LIN {X -0.001,Y -382.805,Z 1558.938,A 0.000,B 0.000,C 90.000,E1 24.771} C_DIS
LIN {X -0.047,Y -376.109,Z 1558.911,A 0.000,B 0.000,C 90.000,E1 20.066} C_DIS
LIN {X -0.062,Y -373.639,Z 1558.897,A 0.000,B 0.000,C 90.000,E1 17.511} C_DIS
LIN {X -0.033,Y -368.037,Z 1558.869,A 0.000,B 0.000,C 90.000,E1 12.355} C_DIS
LIN {X 0.200,Y -366.337,Z 1558.854,A 0.000,B 0.000,C 90.000,E1 9.726} C_DIS
LIN {X 0.078,Y -361.715,Z 1558.821,A 0.000,B 0.000,C 90.000,E1 3.784} C_DIS
LIN {X -0.036,Y -360.828,Z 1558.800,A 0.000,B 0.000,C 90.000,E1 0.057} C_DIS
LIN {X -0.053,Y -359.426,Z 1558.770,A 0.000,B 0.000,C 90.000,E1 354.546} C_DIS
LIN {X 0.070,Y -358.890,Z 1558.759,A 0.000,B 0.000,C 90.000,E1 352.648} C_DIS
LIN {X -0.020,Y -359.563,Z 1558.726,A 0.000,B 0.000,C 90.000,E1 346.645} C_DIS
LIN {X 0.001,Y -361.801,Z 1558.684,A 0.000,B 0.000,C 90.000,E1 339.135} C_DIS
LIN {X -0.154,Y -362.053,Z 1558.680,A 0.000,B 0.000,C 90.000,E1 338.411} C_DIS
LIN {X 0.189,Y -365.980,Z 1558.643,A 0.000,B 0.000,C 90.000,E1 331.641} C_DIS
LIN {X 0.029,Y -366.387,Z 1558.639,A 0.000,B 0.000,C 90.000,E1 330.923} C_DIS
LIN {X -0.031,Y -371.355,Z 1558.604,A 0.000,B 0.000,C 90.000,E1 324.642} C_DIS
LIN {X -0.043,Y -371.766,Z 1558.602,A 0.000,B 0.000,C 90.000,E1 324.276} C_DIS
LIN {X 0.013,Y -377.358,Z 1558.567,A 0.000,B 0.000,C 90.000,E1 318.038} C_DIS
LIN {X 0.012,Y -378.235,Z 1558.563,A 0.000,B 0.000,C 90.000,E1 317.310} C_DIS
LIN {X 0.002,Y -383.940,Z 1558.531,A 0.000,B 0.000,C 90.000,E1 311.515} C_DIS
LIN {X 0.088,Y -384.893,Z 1558.527,A 0.000,B 0.000,C 90.000,E1 310.782} C_DIS
LIN {X 0.262,Y -390.610,Z 1558.495,A 0.000,B 0.000,C 90.000,E1 305.025} C_DIS
LIN {X 0.106,Y -391.104,Z 1558.493,A 0.000,B 0.000,C 90.000,E1 304.692} C_DIS
LIN {X 0.022,Y -391.648,Z 1558.489,A 0.000,B 0.000,C 90.000,E1 303.992} C_DIS
LIN {X -0.080,Y -396.825,Z 1558.459,A 0.000,B 0.000,C 90.000,E1 298.693} C_DIS
LIN {X -0.210,Y -397.120,Z 1558.457,A 0.000,B 0.000,C 90.000,E1 298.359} C_DIS
LIN {X -0.055,Y -401.597,Z 1558.426,A 0.000,B 0.000,C 90.000,E1 292.717} C_DIS
LIN {X 0.222,Y -404.659,Z 1558.395,A 0.000,B 0.000,C 90.000,E1 287.094} C_DIS
LIN {X -0.079,Y -404.735,Z 1558.391,A 0.000,B 0.000,C 90.000,E1 286.441} C_DIS
LIN {X 0.214,Y -406.099,Z 1558.364,A 0.000,B 0.000,C 90.000,E1 281.535} C_DIS
LIN {X -0.176,Y -406.094,Z 1558.362,A 0.000,B 0.000,C 90.000,E1 281.243} C_DIS
LIN {X -0.097,Y -405.680,Z 1558.333,A 0.000,B 0.000,C 90.000,E1 276.024} C_DIS
LIN {X -0.165,Y -405.058,Z 1558.328,A 0.000,B 0.000,C 90.000,E1 274.992} C_DIS
LIN {X -0.060,Y -403.497,Z 1558.304,A 0.000,B 0.000,C 90.000,E1 270.802} C_DIS
LIN {X -0.092,Y -403.288,Z 1558.302,A 0.000,B 0.000,C 90.000,E1 270.458} C_DIS
LIN {X 0.091,Y -398.931,Z 1558.271,A 0.000,B 0.000,C 90.000,E1 264.837} C_DIS
LIN {X -0.040,Y -393.108,Z 1558.242,A 0.000,B 0.000,C 90.000,E1 259.567} C_DIS
LIN {X -0.079,Y -392.835,Z 1558.240,A 0.000,B 0.000,C 90.000,E1 259.218} C_DIS
LIN {X 0.034,Y -385.993,Z 1558.212,A 0.000,B 0.000,C 90.000,E1 254.212} C_DIS
LIN {X -0.026,Y -385.267,Z 1558.208,A 0.000,B 0.000,C 90.000,E1 253.504} C_DIS
LIN {X -0.004,Y -384.768,Z 1558.206,A 0.000,B 0.000,C 90.000,E1 253.142} C_DIS
LIN {X 0.221,Y -377.973,Z 1558.182,A 0.000,B 0.000,C 90.000,E1 248.773} C_DIS
LIN {X -0.044,Y -376.233,Z 1558.174,A 0.000,B 0.000,C 90.000,E1 247.358} C_DIS
LIN {X 0.057,Y -374.944,Z 1558.170,A 0.000,B 0.000,C 90.000,E1 246.613} C_DIS
LIN {X -0.208,Y -368.417,Z 1558.148,A 0.000,B 0.000,C 90.000,E1 242.615} C_DIS
LIN {X 0.097,Y -366.047,Z 1558.137,A 0.000,B 0.000,C 90.000,E1 240.717} C_DIS
LIN {X 0.004,Y -359.196,Z 1558.115,A 0.000,B 0.000,C 90.000,E1 236.628} C_DIS
LIN {X 0.021,Y -355.842,Z 1558.100,A 0.000,B 0.000,C 90.000,E1 233.989} C_DIS
LIN {X -0.173,Y -348.793,Z 1558.075,A 0.000,B 0.000,C 90.000,E1 229.461} C_DIS
LIN {X -0.097,Y -346.185,Z 1558.062,A 0.000,B 0.000,C 90.000,E1 227.148} C_DIS
LIN {X -0.088,Y -345.065,Z 1558.058,A 0.000,B 0.000,C 90.000,E1 226.377} C_DIS
LIN {X 0.094,Y -338.586,Z 1558.030,A 0.000,B 0.000,C 90.000,E1 221.310} C_DIS
LIN {X 0.094,Y -336.840,Z 1558.019,A 0.000,B 0.000,C 90.000,E1 219.358} C_DIS
LIN {X 0.014,Y -330.861,Z 1557.988,A 0.000,B 0.000,C 90.000,E1 213.865} C_DIS
LIN {X 0.149,Y -329.296,Z 1557.975,A 0.000,B 0.000,C 90.000,E1 211.465} C_DIS
LIN {X -0.154,Y -324.669,Z 1557.942,A 0.000,B 0.000,C 90.000,E1 205.540} C_DIS
LIN {X 0.174,Y -323.837,Z 1557.928,A 0.000,B 0.000,C 90.000,E1 203.078} C_DIS
LIN {X -0.017,Y -321.124,Z 1557.881,A 0.000,B 0.000,C 90.000,E1 194.662} C_DIS
LIN {X 0.138,Y -320.932,Z 1557.877,A 0.000,B 0.000,C 90.000,E1 193.828} C_DIS
LIN {X -0.076,Y -321.562,Z 1557.832,A 0.000,B 0.000,C 90.000,E1 185.796} C_DIS
LIN {X -0.143,Y -324.415,Z 1557.790,A 0.000,B 0.000,C 90.000,E1 178.165} C_DIS
LIN {X -0.141,Y -325.376,Z 1557.783,A 0.000,B 0.000,C 90.000,E1 176.963} C_DIS
LIN {X -0.100,Y -329.112,Z 1557.750,A 0.000,B 0.000,C 90.000,E1 170.971} C_DIS
LIN {X 0.061,Y -334.260,Z 1557.726,A 0.000,B 0.000,C 90.000,E1 166.589} C_DIS
LIN {X 0.067,Y -335.488,Z 1557.719,A 0.000,B 0.000,C 90.000,E1 165.408} C_DIS
LIN {X 0.143,Y -340.932,Z 1557.695,A 0.000,B 0.000,C 90.000,E1 161.094} C_DIS
LIN {X -0.172,Y -342.138,Z 1557.691,A 0.000,B 0.000,C 90.000,E1 160.369} C_DIS
LIN {X -0.058,Y -347.939,Z 1557.667,A 0.000,B 0.000,C 90.000,E1 156.102} C_DIS
LIN {X -0.081,Y -354.259,Z 1557.648,A 0.000,B 0.000,C 90.000,E1 152.666} C_DIS
LIN {X -0.222,Y -361.406,Z 1557.625,A 0.000,B 0.000,C 90.000,E1 148.535} C_DIS
LIN {X 0.065,Y -368.758,Z 1557.606,A 0.000,B 0.000,C 90.000,E1 145.135} C_DIS
LIN {X 0.065,Y -377.029,Z 1557.584,A 0.000,B 0.000,C 90.000,E1 141.090} C_DIS
LIN {X -0.061,Y -383.435,Z 1557.570,A 0.000,B 0.000,C 90.000,E1 138.566} C_DIS
LIN {X -0.015,Y -385.037,Z 1557.566,A 0.000,B 0.000,C 90.000,E1 137.838} C_DIS
LIN {X -0.004,Y -394.325,Z 1557.544,A 0.000,B 0.000,C 90.000,E1 133.905} C_DIS
LIN {X 0.107,Y -399.276,Z 1557.534,A 0.000,B 0.000,C 90.000,E1 132.123} C_DIS
LIN {X 0.210,Y -400.192,Z 1557.532,A 0.000,B 0.000,C 90.000,E1 131.757} C_DIS
LIN {X -0.113,Y -409.687,Z 1557.511,A 0.000,B 0.000,C 90.000,E1 127.971} C_DIS
LIN {X 0.046,Y -415.746,Z 1557.499,A 0.000,B 0.000,C 90.000,E1 125.884} C_DIS
LIN {X 0.153,Y -425.188,Z 1557.479,A 0.000,B 0.000,C 90.000,E1 122.133} C_DIS
LIN {X 0.087,Y -430.186,Z 1557.469,A 0.000,B 0.000,C 90.000,E1 120.463} C_DIS
LIN {X 0.086,Y -431.107,Z 1557.468,A 0.000,B 0.000,C 90.000,E1 120.129} C_DIS
LIN {X 0.213,Y -432.689,Z 1557.464,A 0.000,B 0.000,C 90.000,E1 119.411} C_DIS
LIN {X 0.235,Y -547.529,Z 1557.464,A 0.000,B 0.000,C 90.000,E1 119.411} C_DIS
LIN {X 0.136,Y -547.944,Z 1557.464,A 0.000,B 0.000,C 90.000,E1 119.411} C_DIS
LIN {X -0.002,Y -549.482,Z 1557.463,A 0.000,B 0.000,C 90.000,E1 119.283} C_DIS
LIN {X -0.140,Y -550.297,Z 1557.462,A 0.000,B 0.000,C 90.000,E1 119.155} C_DIS
LIN {X -0.113,Y -551.406,Z 1557.460,A 0.000,B 0.000,C 90.000,E1 118.871} C_DIS
LIN {X 0.136,Y -552.267,Z 1557.459,A 0.000,B 0.000,C 90.000,E1 118.565} C_DIS
LIN {X -0.095,Y -552.986,Z 1557.457,A 0.000,B 0.000,C 90.000,E1 118.309} C_DIS
LIN {X 0.202,Y -554.083,Z 1557.454,A 0.000,B 0.000,C 90.000,E1 117.719} C_DIS
LIN {X 0.286,Y -555.333,Z 1557.449,A 0.000,B 0.000,C 90.000,E1 116.873} C_DIS
LIN {X 0.132,Y -556.264,Z 1557.445,A 0.000,B 0.000,C 90.000,E1 116.052} C_DIS
LIN {X 0.232,Y -556.929,Z 1557.440,A 0.000,B 0.000,C 90.000,E1 115.207} C_DIS
LIN {X 0.095,Y -557.406,Z 1557.436,A 0.000,B 0.000,C 90.000,E1 114.387} C_DIS
LIN {X 0.259,Y -557.817,Z 1557.429,A 0.000,B 0.000,C 90.000,E1 113.259} C_DIS
LIN {X 0.295,Y -558.115,Z 1557.420,A 0.000,B 0.000,C 90.000,E1 111.589} C_DIS
LIN {X 0.254,Y -558.382,Z 1557.414,A 0.000,B 0.000,C 90.000,E1 110.482} C_DIS
LIN {X 0.214,Y -558.672,Z 1557.403,A 0.000,B 0.000,C 90.000,E1 108.544} C_DIS
LIN {X 0.014,Y -559.067,Z 1557.392,A 0.000,B 0.000,C 90.000,E1 106.622} C_DIS
LIN {X 0.206,Y -559.382,Z 1557.382,A 0.000,B 0.000,C 90.000,E1 104.662} C_DIS
LIN {X -0.130,Y -559.748,Z 1557.369,A 0.000,B 0.000,C 90.000,E1 102.479} C_DIS
LIN {X -0.186,Y -560.141,Z 1557.359,A 0.000,B 0.000,C 90.000,E1 100.546} C_DIS
LIN {X 0.060,Y -560.700,Z 1557.349,A 0.000,B 0.000,C 90.000,E1 98.859} C_DIS
LIN {X 0.085,Y -561.063,Z 1557.342,A 0.000,B 0.000,C 90.000,E1 97.473} C_DIS
LIN {X -0.212,Y -561.574,Z 1557.331,A 0.000,B 0.000,C 90.000,E1 95.568} C_DIS
LIN {X -0.094,Y -562.028,Z 1557.322,A 0.000,B 0.000,C 90.000,E1 93.898} C_DIS
LIN {X 0.057,Y -562.524,Z 1557.311,A 0.000,B 0.000,C 90.000,E1 91.949} C_DIS
LIN {X 0.124,Y -562.968,Z 1557.302,A 0.000,B 0.000,C 90.000,E1 90.286} C_DIS
LIN {X -0.274,Y -563.518,Z 1557.291,A 0.000,B 0.000,C 90.000,E1 88.396} C_DIS
LIN {X 0.265,Y -563.992,Z 1557.283,A 0.000,B 0.000,C 90.000,E1 86.963} C_DIS
LIN {X -0.030,Y -564.769,Z 1557.273,A 0.000,B 0.000,C 90.000,E1 85.065} C_DIS
LIN {X 0.262,Y -565.685,Z 1557.262,A 0.000,B 0.000,C 90.000,E1 83.109} C_DIS
LIN {X -0.021,Y -566.590,Z 1557.253,A 0.000,B 0.000,C 90.000,E1 81.489} C_DIS
LIN {X 0.193,Y -567.568,Z 1557.245,A 0.000,B 0.000,C 90.000,E1 80.095} C_DIS
LIN {X -0.152,Y -569.200,Z 1557.233,A 0.000,B 0.000,C 90.000,E1 77.937} C_DIS
LIN {X 0.207,Y -570.273,Z 1557.225,A 0.000,B 0.000,C 90.000,E1 76.533} C_DIS
LIN {X 0.160,Y -571.223,Z 1557.218,A 0.000,B 0.000,C 90.000,E1 75.172} C_DIS
LIN {X -0.098,Y -572.486,Z 1557.206,A 0.000,B 0.000,C 90.000,E1 73.015} C_DIS
LIN {X -0.311,Y -573.388,Z 1557.197,A 0.000,B 0.000,C 90.000,E1 71.402} C_DIS
LIN {X 0.032,Y -574.192,Z 1557.189,A 0.000,B 0.000,C 90.000,E1 70.007} C_DIS
LIN {X -0.321,Y -575.150,Z 1557.180,A 0.000,B 0.000,C 90.000,E1 68.411} C_DIS
LIN {X -0.062,Y -576.417,Z 1557.169,A 0.000,B 0.000,C 90.000,E1 66.485} C_DIS
LIN {X 0.085,Y -577.433,Z 1557.160,A 0.000,B 0.000,C 90.000,E1 64.845} C_DIS
LIN {X 0.102,Y -578.606,Z 1557.150,A 0.000,B 0.000,C 90.000,E1 62.948} C_DIS
LIN {X 0.299,Y -579.699,Z 1557.141,A 0.000,B 0.000,C 90.000,E1 61.307} C_DIS
LIN {X 0.018,Y -580.309,Z 1557.135,A 0.000,B 0.000,C 90.000,E1 60.255} C_DIS
LIN {X -0.258,Y -580.520,Z 1557.129,A 0.000,B 0.000,C 90.000,E1 59.203} C_DIS
LIN {X -0.234,Y -580.505,Z 1557.123,A 0.000,B 0.000,C 90.000,E1 58.122} C_DIS
LIN {X -0.222,Y -580.344,Z 1557.120,A 0.000,B 0.000,C 90.000,E1 57.582} C_DIS
LIN {X -0.211,Y -579.942,Z 1557.117,A 0.000,B 0.000,C 90.000,E1 57.041} C_DIS
LIN {X -0.204,Y -579.166,Z 1557.114,A 0.000,B 0.000,C 90.000,E1 56.501} C_DIS
LIN {X -0.043,Y -578.534,Z 1557.112,A 0.000,B 0.000,C 90.000,E1 56.215} C_DIS
LIN {X -0.180,Y -577.252,Z 1557.111,A 0.000,B 0.000,C 90.000,E1 55.928} C_DIS
LIN {X 0.268,Y -576.550,Z 1557.110,A 0.000,B 0.000,C 90.000,E1 55.801} C_DIS
LIN {X -0.134,Y -575.785,Z 1557.110,A 0.000,B 0.000,C 90.000,E1 55.801} C_DIS
LIN {X -0.134,Y -442.133,Z 1557.110,A 0.000,B 0.000,C 90.000,E1 55.801} C_DIS
LIN {X 0.137,Y -433.157,Z 1557.087,A 0.000,B 0.000,C 90.000,E1 51.698} C_DIS
LIN {X -0.023,Y -431.283,Z 1557.082,A 0.000,B 0.000,C 90.000,E1 50.723} C_DIS
LIN {X -0.019,Y -422.094,Z 1557.059,A 0.000,B 0.000,C 90.000,E1 46.701} C_DIS
LIN {X 0.050,Y -418.963,Z 1557.050,A 0.000,B 0.000,C 90.000,E1 45.000} C_DIS
LIN {X -0.062,Y -418.275,Z 1557.048,A 0.000,B 0.000,C 90.000,E1 44.676} C_DIS
LIN {X 0.014,Y -408.785,Z 1557.023,A 0.000,B 0.000,C 90.000,E1 40.216} C_DIS
LIN {X 0.188,Y -405.869,Z 1557.014,A 0.000,B 0.000,C 90.000,E1 38.463} C_DIS
LIN {X -0.163,Y -397.556,Z 1556.991,A 0.000,B 0.000,C 90.000,E1 34.326} C_DIS
LIN {X 0.245,Y -393.794,Z 1556.977,A 0.000,B 0.000,C 90.000,E1 31.799} C_DIS
LIN {X -0.174,Y -386.377,Z 1556.953,A 0.000,B 0.000,C 90.000,E1 27.590} C_DIS
LIN {X -0.032,Y -382.670,Z 1556.937,A 0.000,B 0.000,C 90.000,E1 24.695} C_DIS
LIN {X -0.099,Y -376.018,Z 1556.911,A 0.000,B 0.000,C 90.000,E1 19.993} C_DIS
LIN {X 0.118,Y -373.550,Z 1556.897,A 0.000,B 0.000,C 90.000,E1 17.402} C_DIS
LIN {X 0.156,Y -367.973,Z 1556.868,A 0.000,B 0.000,C 90.000,E1 12.243} C_DIS
LIN {X 0.175,Y -366.548,Z 1556.856,A 0.000,B 0.000,C 90.000,E1 10.018} C_DIS
LIN {X -0.113,Y -365.837,Z 1556.852,A 0.000,B 0.000,C 90.000,E1 9.321} C_DIS
LIN {X -0.098,Y -361.396,Z 1556.817,A 0.000,B 0.000,C 90.000,E1 2.980} C_DIS
LIN {X -0.007,Y -360.906,Z 1556.802,A 0.000,B 0.000,C 90.000,E1 0.344} C_DIS
LIN {X 0.105,Y -360.314,Z 1556.795,A 0.000,B 0.000,C 90.000,E1 359.026} C_DIS
LIN {X -0.053,Y -359.426,Z 1556.770,A 0.000,B 0.000,C 90.000,E1 354.546} C_DIS
LIN {X 0.070,Y -358.890,Z 1556.759,A 0.000,B 0.000,C 90.000,E1 352.648} C_DIS
LIN {X -0.020,Y -359.563,Z 1556.726,A 0.000,B 0.000,C 90.000,E1 346.645} C_DIS
LIN {X 0.001,Y -361.801,Z 1556.684,A 0.000,B 0.000,C 90.000,E1 339.135} C_DIS
LIN {X -0.154,Y -362.053,Z 1556.680,A 0.000,B 0.000,C 90.000,E1 338.411} C_DIS
LIN {X 0.189,Y -365.980,Z 1556.643,A 0.000,B 0.000,C 90.000,E1 331.641} C_DIS
LIN {X 0.029,Y -366.387,Z 1556.639,A 0.000,B 0.000,C 90.000,E1 330.923} C_DIS
LIN {X -0.031,Y -371.355,Z 1556.604,A 0.000,B 0.000,C 90.000,E1 324.642} C_DIS
LIN {X -0.043,Y -371.766,Z 1556.602,A 0.000,B 0.000,C 90.000,E1 324.276} C_DIS
LIN {X 0.013,Y -377.358,Z 1556.567,A 0.000,B 0.000,C 90.000,E1 318.038} C_DIS
LIN {X 0.012,Y -378.235,Z 1556.563,A 0.000,B 0.000,C 90.000,E1 317.310} C_DIS
LIN {X 0.002,Y -383.940,Z 1556.531,A 0.000,B 0.000,C 90.000,E1 311.515} C_DIS
LIN {X 0.088,Y -384.893,Z 1556.527,A 0.000,B 0.000,C 90.000,E1 310.782} C_DIS
LIN {X 0.262,Y -390.610,Z 1556.495,A 0.000,B 0.000,C 90.000,E1 305.025} C_DIS
LIN {X 0.106,Y -391.104,Z 1556.493,A 0.000,B 0.000,C 90.000,E1 304.692} C_DIS
LIN {X 0.022,Y -391.648,Z 1556.489,A 0.000,B 0.000,C 90.000,E1 303.992} C_DIS
LIN {X -0.080,Y -396.825,Z 1556.459,A 0.000,B 0.000,C 90.000,E1 298.693} C_DIS
LIN {X -0.210,Y -397.120,Z 1556.457,A 0.000,B 0.000,C 90.000,E1 298.359} C_DIS
LIN {X -0.055,Y -401.597,Z 1556.426,A 0.000,B 0.000,C 90.000,E1 292.717} C_DIS
LIN {X 0.222,Y -404.659,Z 1556.395,A 0.000,B 0.000,C 90.000,E1 287.094} C_DIS
LIN {X -0.079,Y -404.735,Z 1556.391,A 0.000,B 0.000,C 90.000,E1 286.441} C_DIS
LIN {X 0.214,Y -406.099,Z 1556.364,A 0.000,B 0.000,C 90.000,E1 281.535} C_DIS
LIN {X -0.176,Y -406.094,Z 1556.362,A 0.000,B 0.000,C 90.000,E1 281.243} C_DIS
LIN {X -0.097,Y -405.680,Z 1556.333,A 0.000,B 0.000,C 90.000,E1 276.024} C_DIS
LIN {X -0.165,Y -405.058,Z 1556.328,A 0.000,B 0.000,C 90.000,E1 274.992} C_DIS
LIN {X -0.060,Y -403.497,Z 1556.304,A 0.000,B 0.000,C 90.000,E1 270.802} C_DIS
LIN {X -0.092,Y -403.288,Z 1556.302,A 0.000,B 0.000,C 90.000,E1 270.458} C_DIS
LIN {X 0.091,Y -398.931,Z 1556.271,A 0.000,B 0.000,C 90.000,E1 264.837} C_DIS
LIN {X -0.040,Y -393.108,Z 1556.242,A 0.000,B 0.000,C 90.000,E1 259.567} C_DIS
LIN {X -0.079,Y -392.835,Z 1556.240,A 0.000,B 0.000,C 90.000,E1 259.218} C_DIS
LIN {X 0.034,Y -385.993,Z 1556.212,A 0.000,B 0.000,C 90.000,E1 254.212} C_DIS
LIN {X -0.026,Y -385.267,Z 1556.208,A 0.000,B 0.000,C 90.000,E1 253.504} C_DIS
LIN {X -0.004,Y -384.768,Z 1556.206,A 0.000,B 0.000,C 90.000,E1 253.142} C_DIS
LIN {X 0.221,Y -377.973,Z 1556.182,A 0.000,B 0.000,C 90.000,E1 248.773} C_DIS
LIN {X -0.044,Y -376.233,Z 1556.174,A 0.000,B 0.000,C 90.000,E1 247.358} C_DIS
LIN {X 0.057,Y -374.944,Z 1556.170,A 0.000,B 0.000,C 90.000,E1 246.613} C_DIS
LIN {X -0.208,Y -368.417,Z 1556.148,A 0.000,B 0.000,C 90.000,E1 242.615} C_DIS
LIN {X 0.097,Y -366.047,Z 1556.137,A 0.000,B 0.000,C 90.000,E1 240.717} C_DIS
LIN {X 0.004,Y -359.196,Z 1556.115,A 0.000,B 0.000,C 90.000,E1 236.628} C_DIS
LIN {X 0.021,Y -355.842,Z 1556.100,A 0.000,B 0.000,C 90.000,E1 233.989} C_DIS
LIN {X -0.173,Y -348.793,Z 1556.075,A 0.000,B 0.000,C 90.000,E1 229.461} C_DIS
LIN {X -0.097,Y -346.185,Z 1556.062,A 0.000,B 0.000,C 90.000,E1 227.148} C_DIS
LIN {X -0.088,Y -345.065,Z 1556.058,A 0.000,B 0.000,C 90.000,E1 226.377} C_DIS
LIN {X 0.094,Y -338.586,Z 1556.030,A 0.000,B 0.000,C 90.000,E1 221.310} C_DIS
LIN {X 0.094,Y -336.840,Z 1556.019,A 0.000,B 0.000,C 90.000,E1 219.358} C_DIS
LIN {X 0.014,Y -330.861,Z 1555.988,A 0.000,B 0.000,C 90.000,E1 213.865} C_DIS
LIN {X 0.149,Y -329.296,Z 1555.975,A 0.000,B 0.000,C 90.000,E1 211.465} C_DIS
LIN {X -0.154,Y -324.669,Z 1555.942,A 0.000,B 0.000,C 90.000,E1 205.540} C_DIS
LIN {X 0.174,Y -323.837,Z 1555.928,A 0.000,B 0.000,C 90.000,E1 203.078} C_DIS
LIN {X -0.017,Y -321.124,Z 1555.881,A 0.000,B 0.000,C 90.000,E1 194.662} C_DIS
LIN {X 0.138,Y -320.932,Z 1555.877,A 0.000,B 0.000,C 90.000,E1 193.828} C_DIS
LIN {X -0.076,Y -321.562,Z 1555.832,A 0.000,B 0.000,C 90.000,E1 185.796} C_DIS
LIN {X -0.143,Y -324.415,Z 1555.790,A 0.000,B 0.000,C 90.000,E1 178.165} C_DIS
LIN {X -0.141,Y -325.376,Z 1555.783,A 0.000,B 0.000,C 90.000,E1 176.963} C_DIS
LIN {X -0.100,Y -329.112,Z 1555.750,A 0.000,B 0.000,C 90.000,E1 170.971} C_DIS
LIN {X 0.061,Y -334.260,Z 1555.726,A 0.000,B 0.000,C 90.000,E1 166.589} C_DIS
LIN {X 0.067,Y -335.488,Z 1555.719,A 0.000,B 0.000,C 90.000,E1 165.408} C_DIS
LIN {X 0.143,Y -340.932,Z 1555.695,A 0.000,B 0.000,C 90.000,E1 161.094} C_DIS
LIN {X -0.172,Y -342.138,Z 1555.691,A 0.000,B 0.000,C 90.000,E1 160.369} C_DIS
LIN {X -0.058,Y -347.939,Z 1555.667,A 0.000,B 0.000,C 90.000,E1 156.102} C_DIS
LIN {X -0.081,Y -354.259,Z 1555.648,A 0.000,B 0.000,C 90.000,E1 152.666} C_DIS
LIN {X -0.222,Y -361.406,Z 1555.625,A 0.000,B 0.000,C 90.000,E1 148.535} C_DIS
LIN {X 0.065,Y -368.758,Z 1555.606,A 0.000,B 0.000,C 90.000,E1 145.135} C_DIS
LIN {X 0.065,Y -377.029,Z 1555.584,A 0.000,B 0.000,C 90.000,E1 141.090} C_DIS
LIN {X -0.061,Y -383.435,Z 1555.570,A 0.000,B 0.000,C 90.000,E1 138.566} C_DIS
LIN {X -0.015,Y -385.037,Z 1555.566,A 0.000,B 0.000,C 90.000,E1 137.838} C_DIS
LIN {X -0.004,Y -394.325,Z 1555.544,A 0.000,B 0.000,C 90.000,E1 133.905} C_DIS
LIN {X 0.107,Y -399.276,Z 1555.534,A 0.000,B 0.000,C 90.000,E1 132.123} C_DIS
LIN {X 0.210,Y -400.192,Z 1555.532,A 0.000,B 0.000,C 90.000,E1 131.757} C_DIS
LIN {X -0.113,Y -409.687,Z 1555.511,A 0.000,B 0.000,C 90.000,E1 127.971} C_DIS
LIN {X 0.046,Y -415.746,Z 1555.499,A 0.000,B 0.000,C 90.000,E1 125.884} C_DIS
LIN {X 0.153,Y -425.188,Z 1555.479,A 0.000,B 0.000,C 90.000,E1 122.133} C_DIS
LIN {X -0.021,Y -429.348,Z 1555.471,A 0.000,B 0.000,C 90.000,E1 120.747} C_DIS
LIN {X -0.059,Y -547.338,Z 1555.471,A 0.000,B 0.000,C 90.000,E1 120.747} C_DIS
LIN {X 0.189,Y -547.525,Z 1555.471,A 0.000,B 0.000,C 90.000,E1 120.718} C_DIS
LIN {X 0.151,Y -549.162,Z 1555.470,A 0.000,B 0.000,C 90.000,E1 120.590} C_DIS
LIN {X 0.111,Y -549.962,Z 1555.469,A 0.000,B 0.000,C 90.000,E1 120.463} C_DIS
LIN {X -0.132,Y -551.149,Z 1555.468,A 0.000,B 0.000,C 90.000,E1 120.207} C_DIS
LIN {X -0.095,Y -552.015,Z 1555.466,A 0.000,B 0.000,C 90.000,E1 119.922} C_DIS
LIN {X 0.191,Y -553.358,Z 1555.463,A 0.000,B 0.000,C 90.000,E1 119.333} C_DIS
LIN {X 0.265,Y -554.779,Z 1555.458,A 0.000,B 0.000,C 90.000,E1 118.487} C_DIS
LIN {X 0.355,Y -555.806,Z 1555.454,A 0.000,B 0.000,C 90.000,E1 117.641} C_DIS
LIN {X -0.011,Y -556.785,Z 1555.448,A 0.000,B 0.000,C 90.000,E1 116.565} C_DIS
LIN {X -0.114,Y -557.426,Z 1555.441,A 0.000,B 0.000,C 90.000,E1 115.463} C_DIS
LIN {X 0.051,Y -557.781,Z 1555.435,A 0.000,B 0.000,C 90.000,E1 114.335} C_DIS
LIN {X 0.224,Y -558.098,Z 1555.429,A 0.000,B 0.000,C 90.000,E1 113.206} C_DIS
LIN {X -0.247,Y -558.383,Z 1555.420,A 0.000,B 0.000,C 90.000,E1 111.589} C_DIS
LIN {X 0.240,Y -558.636,Z 1555.414,A 0.000,B 0.000,C 90.000,E1 110.429} C_DIS
LIN {X 0.213,Y -558.948,Z 1555.403,A 0.000,B 0.000,C 90.000,E1 108.489} C_DIS
LIN {X 0.025,Y -559.341,Z 1555.392,A 0.000,B 0.000,C 90.000,E1 106.567} C_DIS
LIN {X -0.171,Y -559.638,Z 1555.381,A 0.000,B 0.000,C 90.000,E1 104.647} C_DIS
LIN {X 0.025,Y -560.013,Z 1555.369,A 0.000,B 0.000,C 90.000,E1 102.411} C_DIS
LIN {X 0.009,Y -560.494,Z 1555.357,A 0.000,B 0.000,C 90.000,E1 100.197} C_DIS
LIN {X 0.114,Y -560.999,Z 1555.349,A 0.000,B 0.000,C 90.000,E1 98.803} C_DIS
LIN {X 0.219,Y -561.348,Z 1555.341,A 0.000,B 0.000,C 90.000,E1 97.409} C_DIS
LIN {X -0.226,Y -561.806,Z 1555.332,A 0.000,B 0.000,C 90.000,E1 95.796} C_DIS
LIN {X -0.147,Y -562.298,Z 1555.323,A 0.000,B 0.000,C 90.000,E1 94.131} C_DIS
LIN {X -0.056,Y -562.701,Z 1555.314,A 0.000,B 0.000,C 90.000,E1 92.465} C_DIS
LIN {X 0.012,Y -563.178,Z 1555.305,A 0.000,B 0.000,C 90.000,E1 90.802} C_DIS
LIN {X 0.080,Y -563.627,Z 1555.295,A 0.000,B 0.000,C 90.000,E1 89.141} C_DIS
LIN {X 0.169,Y -564.220,Z 1555.286,A 0.000,B 0.000,C 90.000,E1 87.478} C_DIS
LIN {X -0.159,Y -564.916,Z 1555.275,A 0.000,B 0.000,C 90.000,E1 85.584} C_DIS
LIN {X 0.039,Y -565.685,Z 1555.266,A 0.000,B 0.000,C 90.000,E1 83.913} C_DIS
LIN {X -0.142,Y -566.739,Z 1555.256,A 0.000,B 0.000,C 90.000,E1 82.008} C_DIS
LIN {X -0.223,Y -568.037,Z 1555.245,A 0.000,B 0.000,C 90.000,E1 80.095} C_DIS
LIN {X 0.000,Y -569.642,Z 1555.233,A 0.000,B 0.000,C 90.000,E1 77.881} C_DIS
LIN {X 0.180,Y -570.512,Z 1555.227,A 0.000,B 0.000,C 90.000,E1 76.769} C_DIS
LIN {X -0.230,Y -571.698,Z 1555.218,A 0.000,B 0.000,C 90.000,E1 75.172} C_DIS
LIN {X 0.073,Y -572.947,Z 1555.205,A 0.000,B 0.000,C 90.000,E1 72.960} C_DIS
LIN {X 0.048,Y -573.889,Z 1555.196,A 0.000,B 0.000,C 90.000,E1 71.329} C_DIS
LIN {X -0.327,Y -574.663,Z 1555.189,A 0.000,B 0.000,C 90.000,E1 70.007} C_DIS
LIN {X 0.076,Y -575.625,Z 1555.180,A 0.000,B 0.000,C 90.000,E1 68.337} C_DIS
LIN {X 0.127,Y -576.900,Z 1555.169,A 0.000,B 0.000,C 90.000,E1 66.433} C_DIS
LIN {X -0.246,Y -577.869,Z 1555.160,A 0.000,B 0.000,C 90.000,E1 64.845} C_DIS
LIN {X 0.045,Y -579.090,Z 1555.150,A 0.000,B 0.000,C 90.000,E1 62.922} C_DIS
LIN {X -0.011,Y -580.172,Z 1555.141,A 0.000,B 0.000,C 90.000,E1 61.307} C_DIS
LIN {X 0.077,Y -581.034,Z 1555.133,A 0.000,B 0.000,C 90.000,E1 59.950} C_DIS
LIN {X -0.040,Y -581.655,Z 1555.126,A 0.000,B 0.000,C 90.000,E1 58.614} C_DIS
LIN {X -0.005,Y -582.001,Z 1555.120,A 0.000,B 0.000,C 90.000,E1 57.533} C_DIS
LIN {X 0.182,Y -581.934,Z 1555.115,A 0.000,B 0.000,C 90.000,E1 56.707} C_DIS
LIN {X -0.284,Y -581.688,Z 1555.112,A 0.000,B 0.000,C 90.000,E1 56.215} C_DIS
LIN {X -0.266,Y -581.170,Z 1555.109,A 0.000,B 0.000,C 90.000,E1 55.674} C_DIS
LIN {X -0.096,Y -580.784,Z 1555.108,A 0.000,B 0.000,C 90.000,E1 55.388} C_DIS
LIN {X 0.075,Y -580.268,Z 1555.106,A 0.000,B 0.000,C 90.000,E1 55.102} C_DIS
LIN {X -0.089,Y -579.468,Z 1555.105,A 0.000,B 0.000,C 90.000,E1 54.848} C_DIS
LIN {X 0.162,Y -578.872,Z 1555.104,A 0.000,B 0.000,C 90.000,E1 54.689} C_DIS
LIN {X 0.078,Y -577.907,Z 1555.103,A 0.000,B 0.000,C 90.000,E1 54.562} C_DIS
LIN {X 0.287,Y -576.938,Z 1555.103,A 0.000,B 0.000,C 90.000,E1 54.482} C_DIS
LIN {X 0.257,Y -576.796,Z 1555.103,A 0.000,B 0.000,C 90.000,E1 54.482} C_DIS
LIN {X 0.171,Y -439.026,Z 1555.103,A 0.000,B 0.000,C 90.000,E1 54.482} C_DIS
LIN {X -0.121,Y -431.829,Z 1555.083,A 0.000,B 0.000,C 90.000,E1 51.009} C_DIS
LIN {X 0.139,Y -431.129,Z 1555.082,A 0.000,B 0.000,C 90.000,E1 50.642} C_DIS
LIN {X 0.135,Y -421.975,Z 1555.059,A 0.000,B 0.000,C 90.000,E1 46.620} C_DIS
LIN {X 0.201,Y -418.859,Z 1555.050,A 0.000,B 0.000,C 90.000,E1 44.919} C_DIS
LIN {X -0.026,Y -417.298,Z 1555.046,A 0.000,B 0.000,C 90.000,E1 44.271} C_DIS
LIN {X 0.043,Y -408.064,Z 1555.021,A 0.000,B 0.000,C 90.000,E1 39.806} C_DIS
LIN {X -0.250,Y -405.741,Z 1555.014,A 0.000,B 0.000,C 90.000,E1 38.463} C_DIS
LIN {X -0.045,Y -397.450,Z 1554.990,A 0.000,B 0.000,C 90.000,E1 34.246} C_DIS
LIN {X -0.188,Y -393.685,Z 1554.977,A 0.000,B 0.000,C 90.000,E1 31.799} C_DIS
LIN {X -0.083,Y -386.285,Z 1554.953,A 0.000,B 0.000,C 90.000,E1 27.513} C_DIS
LIN {X 0.075,Y -383.060,Z 1554.939,A 0.000,B 0.000,C 90.000,E1 24.975} C_DIS
LIN {X 0.044,Y -381.952,Z 1554.935,A 0.000,B 0.000,C 90.000,E1 24.259} C_DIS
LIN {X -0.187,Y -375.551,Z 1554.909,A 0.000,B 0.000,C 90.000,E1 19.577} C_DIS
LIN {X 0.049,Y -373.459,Z 1554.896,A 0.000,B 0.000,C 90.000,E1 17.347} C_DIS
LIN {X 0.092,Y -367.923,Z 1554.868,A 0.000,B 0.000,C 90.000,E1 12.187} C_DIS
LIN {X 0.113,Y -366.515,Z 1554.855,A 0.000,B 0.000,C 90.000,E1 9.962} C_DIS
LIN {X 0.048,Y -361.813,Z 1554.822,A 0.000,B 0.000,C 90.000,E1 4.012} C_DIS
LIN {X -0.067,Y -360.904,Z 1554.802,A 0.000,B 0.000,C 90.000,E1 0.286} C_DIS
LIN {X -0.053,Y -359.426,Z 1554.770,A 0.000,B 0.000,C 90.000,E1 354.546} C_DIS
LIN {X 0.070,Y -358.890,Z 1554.759,A 0.000,B 0.000,C 90.000,E1 352.648} C_DIS
LIN {X -0.020,Y -359.563,Z 1554.726,A 0.000,B 0.000,C 90.000,E1 346.645} C_DIS
LIN {X 0.001,Y -361.801,Z 1554.684,A 0.000,B 0.000,C 90.000,E1 339.135} C_DIS
LIN {X -0.154,Y -362.053,Z 1554.680,A 0.000,B 0.000,C 90.000,E1 338.411} C_DIS
LIN {X 0.189,Y -365.980,Z 1554.643,A 0.000,B 0.000,C 90.000,E1 331.641} C_DIS
LIN {X 0.029,Y -366.387,Z 1554.639,A 0.000,B 0.000,C 90.000,E1 330.923} C_DIS
LIN {X -0.031,Y -371.355,Z 1554.604,A 0.000,B 0.000,C 90.000,E1 324.642} C_DIS
LIN {X -0.043,Y -371.766,Z 1554.602,A 0.000,B 0.000,C 90.000,E1 324.276} C_DIS
LIN {X 0.013,Y -377.358,Z 1554.567,A 0.000,B 0.000,C 90.000,E1 318.038} C_DIS
LIN {X 0.012,Y -378.235,Z 1554.563,A 0.000,B 0.000,C 90.000,E1 317.310} C_DIS
LIN {X 0.002,Y -383.940,Z 1554.531,A 0.000,B 0.000,C 90.000,E1 311.515} C_DIS
LIN {X 0.088,Y -384.893,Z 1554.527,A 0.000,B 0.000,C 90.000,E1 310.782} C_DIS
LIN {X 0.262,Y -390.610,Z 1554.495,A 0.000,B 0.000,C 90.000,E1 305.025} C_DIS
LIN {X 0.106,Y -391.104,Z 1554.493,A 0.000,B 0.000,C 90.000,E1 304.692} C_DIS
LIN {X 0.022,Y -391.648,Z 1554.489,A 0.000,B 0.000,C 90.000,E1 303.992} C_DIS
LIN {X -0.080,Y -396.825,Z 1554.459,A 0.000,B 0.000,C 90.000,E1 298.693} C_DIS
LIN {X -0.210,Y -397.120,Z 1554.457,A 0.000,B 0.000,C 90.000,E1 298.359} C_DIS
LIN {X -0.055,Y -401.597,Z 1554.426,A 0.000,B 0.000,C 90.000,E1 292.717} C_DIS
LIN {X 0.222,Y -404.659,Z 1554.395,A 0.000,B 0.000,C 90.000,E1 287.094} C_DIS
LIN {X -0.079,Y -404.735,Z 1554.391,A 0.000,B 0.000,C 90.000,E1 286.441} C_DIS
LIN {X 0.214,Y -406.099,Z 1554.364,A 0.000,B 0.000,C 90.000,E1 281.535} C_DIS
LIN {X -0.176,Y -406.094,Z 1554.362,A 0.000,B 0.000,C 90.000,E1 281.243} C_DIS
LIN {X -0.097,Y -405.680,Z 1554.333,A 0.000,B 0.000,C 90.000,E1 276.024} C_DIS
LIN {X -0.165,Y -405.058,Z 1554.328,A 0.000,B 0.000,C 90.000,E1 274.992} C_DIS
LIN {X -0.060,Y -403.497,Z 1554.304,A 0.000,B 0.000,C 90.000,E1 270.802} C_DIS
LIN {X -0.092,Y -403.288,Z 1554.302,A 0.000,B 0.000,C 90.000,E1 270.458} C_DIS
LIN {X 0.091,Y -398.931,Z 1554.271,A 0.000,B 0.000,C 90.000,E1 264.837} C_DIS
LIN {X -0.040,Y -393.108,Z 1554.242,A 0.000,B 0.000,C 90.000,E1 259.567} C_DIS
LIN {X -0.079,Y -392.835,Z 1554.240,A 0.000,B 0.000,C 90.000,E1 259.218} C_DIS
LIN {X 0.034,Y -385.993,Z 1554.212,A 0.000,B 0.000,C 90.000,E1 254.212} C_DIS
LIN {X -0.026,Y -385.267,Z 1554.208,A 0.000,B 0.000,C 90.000,E1 253.504} C_DIS
LIN {X -0.004,Y -384.768,Z 1554.206,A 0.000,B 0.000,C 90.000,E1 253.142} C_DIS
LIN {X 0.221,Y -377.973,Z 1554.182,A 0.000,B 0.000,C 90.000,E1 248.773} C_DIS
LIN {X -0.044,Y -376.233,Z 1554.174,A 0.000,B 0.000,C 90.000,E1 247.358} C_DIS
LIN {X 0.057,Y -374.944,Z 1554.170,A 0.000,B 0.000,C 90.000,E1 246.613} C_DIS
LIN {X -0.208,Y -368.417,Z 1554.148,A 0.000,B 0.000,C 90.000,E1 242.615} C_DIS
LIN {X 0.097,Y -366.047,Z 1554.137,A 0.000,B 0.000,C 90.000,E1 240.717} C_DIS
LIN {X 0.004,Y -359.196,Z 1554.115,A 0.000,B 0.000,C 90.000,E1 236.628} C_DIS
LIN {X 0.021,Y -355.842,Z 1554.100,A 0.000,B 0.000,C 90.000,E1 233.989} C_DIS
LIN {X -0.173,Y -348.793,Z 1554.075,A 0.000,B 0.000,C 90.000,E1 229.461} C_DIS
LIN {X -0.097,Y -346.185,Z 1554.062,A 0.000,B 0.000,C 90.000,E1 227.148} C_DIS
LIN {X -0.088,Y -345.065,Z 1554.058,A 0.000,B 0.000,C 90.000,E1 226.377} C_DIS
LIN {X 0.094,Y -338.586,Z 1554.030,A 0.000,B 0.000,C 90.000,E1 221.310} C_DIS
LIN {X 0.094,Y -336.840,Z 1554.019,A 0.000,B 0.000,C 90.000,E1 219.358} C_DIS
LIN {X 0.014,Y -330.861,Z 1553.988,A 0.000,B 0.000,C 90.000,E1 213.865} C_DIS
LIN {X 0.149,Y -329.296,Z 1553.975,A 0.000,B 0.000,C 90.000,E1 211.465} C_DIS
LIN {X -0.154,Y -324.669,Z 1553.942,A 0.000,B 0.000,C 90.000,E1 205.540} C_DIS
LIN {X 0.174,Y -323.837,Z 1553.928,A 0.000,B 0.000,C 90.000,E1 203.078} C_DIS
LIN {X -0.017,Y -321.124,Z 1553.881,A 0.000,B 0.000,C 90.000,E1 194.662} C_DIS
LIN {X 0.138,Y -320.932,Z 1553.877,A 0.000,B 0.000,C 90.000,E1 193.828} C_DIS
LIN {X -0.076,Y -321.562,Z 1553.832,A 0.000,B 0.000,C 90.000,E1 185.796} C_DIS
LIN {X -0.143,Y -324.415,Z 1553.790,A 0.000,B 0.000,C 90.000,E1 178.165} C_DIS
LIN {X -0.141,Y -325.376,Z 1553.783,A 0.000,B 0.000,C 90.000,E1 176.963} C_DIS
LIN {X -0.100,Y -329.112,Z 1553.750,A 0.000,B 0.000,C 90.000,E1 170.971} C_DIS
LIN {X 0.061,Y -334.260,Z 1553.726,A 0.000,B 0.000,C 90.000,E1 166.589} C_DIS
LIN {X 0.067,Y -335.488,Z 1553.719,A 0.000,B 0.000,C 90.000,E1 165.408} C_DIS
LIN {X 0.143,Y -340.932,Z 1553.695,A 0.000,B 0.000,C 90.000,E1 161.094} C_DIS
LIN {X -0.172,Y -342.138,Z 1553.691,A 0.000,B 0.000,C 90.000,E1 160.369} C_DIS
LIN {X -0.058,Y -347.939,Z 1553.667,A 0.000,B 0.000,C 90.000,E1 156.102} C_DIS
LIN {X -0.081,Y -354.259,Z 1553.648,A 0.000,B 0.000,C 90.000,E1 152.666} C_DIS
LIN {X -0.222,Y -361.406,Z 1553.625,A 0.000,B 0.000,C 90.000,E1 148.535} C_DIS
LIN {X 0.065,Y -368.758,Z 1553.606,A 0.000,B 0.000,C 90.000,E1 145.135} C_DIS
LIN {X 0.065,Y -377.029,Z 1553.584,A 0.000,B 0.000,C 90.000,E1 141.090} C_DIS
LIN {X -0.061,Y -383.435,Z 1553.570,A 0.000,B 0.000,C 90.000,E1 138.566} C_DIS
LIN {X -0.015,Y -385.037,Z 1553.566,A 0.000,B 0.000,C 90.000,E1 137.838} C_DIS
LIN {X -0.004,Y -394.325,Z 1553.544,A 0.000,B 0.000,C 90.000,E1 133.905} C_DIS
LIN {X 0.107,Y -399.276,Z 1553.534,A 0.000,B 0.000,C 90.000,E1 132.123} C_DIS
LIN {X 0.210,Y -400.192,Z 1553.532,A 0.000,B 0.000,C 90.000,E1 131.757} C_DIS
LIN {X -0.113,Y -409.687,Z 1553.511,A 0.000,B 0.000,C 90.000,E1 127.971} C_DIS
LIN {X 0.046,Y -415.746,Z 1553.499,A 0.000,B 0.000,C 90.000,E1 125.884} C_DIS
LIN {X 0.174,Y -425.543,Z 1553.478,A 0.000,B 0.000,C 90.000,E1 122.005} C_DIS
LIN {X 0.178,Y -547.471,Z 1553.478,A 0.000,B 0.000,C 90.000,E1 122.005} C_DIS
LIN {X 0.131,Y -547.635,Z 1553.478,A 0.000,B 0.000,C 90.000,E1 122.005} C_DIS
LIN {X 0.169,Y -549.581,Z 1553.477,A 0.000,B 0.000,C 90.000,E1 121.799} C_DIS
LIN {X 0.010,Y -550.799,Z 1553.475,A 0.000,B 0.000,C 90.000,E1 121.544} C_DIS
LIN {X 0.052,Y -551.702,Z 1553.474,A 0.000,B 0.000,C 90.000,E1 121.258} C_DIS
LIN {X -0.141,Y -553.054,Z 1553.471,A 0.000,B 0.000,C 90.000,E1 120.718} C_DIS
LIN {X 0.152,Y -554.079,Z 1553.468,A 0.000,B 0.000,C 90.000,E1 120.129} C_DIS
LIN {X 0.234,Y -555.255,Z 1553.463,A 0.000,B 0.000,C 90.000,E1 119.283} C_DIS
LIN {X 0.116,Y -556.362,Z 1553.457,A 0.000,B 0.000,C 90.000,E1 118.180} C_DIS
LIN {X 0.016,Y -557.060,Z 1553.450,A 0.000,B 0.000,C 90.000,E1 117.078} C_DIS
LIN {X -0.081,Y -557.536,Z 1553.444,A 0.000,B 0.000,C 90.000,E1 115.976} C_DIS
LIN {X -0.210,Y -557.849,Z 1553.440,A 0.000,B 0.000,C 90.000,E1 115.155} C_DIS
LIN {X -0.246,Y -558.257,Z 1553.432,A 0.000,B 0.000,C 90.000,E1 113.770} C_DIS
LIN {X 0.234,Y -558.498,Z 1553.424,A 0.000,B 0.000,C 90.000,E1 112.333} C_DIS
LIN {X -0.131,Y -558.889,Z 1553.413,A 0.000,B 0.000,C 90.000,E1 110.429} C_DIS
LIN {X -0.152,Y -559.222,Z 1553.403,A 0.000,B 0.000,C 90.000,E1 108.489} C_DIS
LIN {X 0.069,Y -559.552,Z 1553.393,A 0.000,B 0.000,C 90.000,E1 106.804} C_DIS
LIN {X 0.132,Y -559.780,Z 1553.384,A 0.000,B 0.000,C 90.000,E1 105.134} C_DIS
LIN {X -0.236,Y -559.949,Z 1553.378,A 0.000,B 0.000,C 90.000,E1 104.064} C_DIS
LIN {X -0.171,Y -560.333,Z 1553.367,A 0.000,B 0.000,C 90.000,E1 102.119} C_DIS
LIN {X 0.123,Y -561.112,Z 1553.352,A 0.000,B 0.000,C 90.000,E1 99.321} C_DIS
LIN {X 0.081,Y -561.468,Z 1553.346,A 0.000,B 0.000,C 90.000,E1 98.219} C_DIS
LIN {X -0.217,Y -562.008,Z 1553.335,A 0.000,B 0.000,C 90.000,E1 96.315} C_DIS
LIN {X -0.090,Y -562.475,Z 1553.326,A 0.000,B 0.000,C 90.000,E1 94.645} C_DIS
LIN {X -0.230,Y -562.787,Z 1553.320,A 0.000,B 0.000,C 90.000,E1 93.555} C_DIS
LIN {X -0.036,Y -563.272,Z 1553.309,A 0.000,B 0.000,C 90.000,E1 91.604} C_DIS
LIN {X -0.077,Y -563.694,Z 1553.301,A 0.000,B 0.000,C 90.000,E1 90.229} C_DIS
LIN {X 0.232,Y -564.422,Z 1553.289,A 0.000,B 0.000,C 90.000,E1 87.993} C_DIS
LIN {X -0.120,Y -565.079,Z 1553.278,A 0.000,B 0.000,C 90.000,E1 86.102} C_DIS
LIN {X 0.175,Y -565.962,Z 1553.268,A 0.000,B 0.000,C 90.000,E1 84.147} C_DIS
LIN {X -0.009,Y -567.014,Z 1553.257,A 0.000,B 0.000,C 90.000,E1 82.243} C_DIS
LIN {X 0.088,Y -568.495,Z 1553.245,A 0.000,B 0.000,C 90.000,E1 80.038} C_DIS
LIN {X 0.137,Y -569.841,Z 1553.234,A 0.000,B 0.000,C 90.000,E1 78.117} C_DIS
LIN {X -0.237,Y -570.762,Z 1553.228,A 0.000,B 0.000,C 90.000,E1 77.061} C_DIS
LIN {X -0.086,Y -571.986,Z 1553.219,A 0.000,B 0.000,C 90.000,E1 75.408} C_DIS
LIN {X 0.053,Y -572.748,Z 1553.211,A 0.000,B 0.000,C 90.000,E1 74.031} C_DIS
LIN {X -0.146,Y -573.719,Z 1553.202,A 0.000,B 0.000,C 90.000,E1 72.417} C_DIS
LIN {X -0.152,Y -574.377,Z 1553.196,A 0.000,B 0.000,C 90.000,E1 71.329} C_DIS
LIN {X 0.218,Y -575.126,Z 1553.189,A 0.000,B 0.000,C 90.000,E1 69.934} C_DIS
LIN {X -0.106,Y -576.091,Z 1553.180,A 0.000,B 0.000,C 90.000,E1 68.337} C_DIS
LIN {X -0.044,Y -577.366,Z 1553.169,A 0.000,B 0.000,C 90.000,E1 66.433} C_DIS
LIN {X -0.030,Y -578.461,Z 1553.159,A 0.000,B 0.000,C 90.000,E1 64.537} C_DIS
LIN {X -0.106,Y -579.558,Z 1553.150,A 0.000,B 0.000,C 90.000,E1 62.922} C_DIS
LIN {X -0.154,Y -580.628,Z 1553.141,A 0.000,B 0.000,C 90.000,E1 61.307} C_DIS
LIN {X -0.057,Y -581.476,Z 1553.133,A 0.000,B 0.000,C 90.000,E1 59.950} C_DIS
LIN {X 0.020,Y -582.825,Z 1553.121,A 0.000,B 0.000,C 90.000,E1 57.788} C_DIS
LIN {X -0.098,Y -583.191,Z 1553.117,A 0.000,B 0.000,C 90.000,E1 56.993} C_DIS
LIN {X 0.102,Y -583.329,Z 1553.112,A 0.000,B 0.000,C 90.000,E1 56.167} C_DIS
LIN {X -0.178,Y -583.151,Z 1553.108,A 0.000,B 0.000,C 90.000,E1 55.388} C_DIS
LIN {X 0.180,Y -582.790,Z 1553.105,A 0.000,B 0.000,C 90.000,E1 54.815} C_DIS
LIN {X 0.198,Y -582.038,Z 1553.102,A 0.000,B 0.000,C 90.000,E1 54.276} C_DIS
LIN {X -0.096,Y -581.546,Z 1553.100,A 0.000,B 0.000,C 90.000,E1 54.036} C_DIS
LIN {X -0.264,Y -580.882,Z 1553.099,A 0.000,B 0.000,C 90.000,E1 53.783} C_DIS
LIN {X -0.046,Y -579.685,Z 1553.097,A 0.000,B 0.000,C 90.000,E1 53.463} C_DIS
LIN {X 0.024,Y -578.731,Z 1553.096,A 0.000,B 0.000,C 90.000,E1 53.336} C_DIS
LIN {X 0.065,Y -578.046,Z 1553.096,A 0.000,B 0.000,C 90.000,E1 53.290} C_DIS
LIN {X -0.029,Y -577.658,Z 1553.096,A 0.000,B 0.000,C 90.000,E1 53.290} C_DIS
LIN {X -0.046,Y -436.309,Z 1553.096,A 0.000,B 0.000,C 90.000,E1 53.290} C_DIS
LIN {X 0.113,Y -431.662,Z 1553.083,A 0.000,B 0.000,C 90.000,E1 50.884} C_DIS
LIN {X 0.101,Y -427.587,Z 1553.074,A 0.000,B 0.000,C 90.000,E1 49.218} C_DIS
LIN {X 0.091,Y -418.693,Z 1553.049,A 0.000,B 0.000,C 90.000,E1 44.838} C_DIS
LIN {X 0.030,Y -409.762,Z 1553.026,A 0.000,B 0.000,C 90.000,E1 40.744} C_DIS
LIN {X 0.053,Y -406.171,Z 1553.015,A 0.000,B 0.000,C 90.000,E1 38.669} C_DIS
LIN {X 0.087,Y -404.738,Z 1553.011,A 0.000,B 0.000,C 90.000,E1 37.971} C_DIS
LIN {X -0.105,Y -396.143,Z 1552.986,A 0.000,B 0.000,C 90.000,E1 33.452} C_DIS
LIN {X 0.135,Y -394.058,Z 1552.978,A 0.000,B 0.000,C 90.000,E1 32.005} C_DIS
LIN {X 0.001,Y -393.484,Z 1552.976,A 0.000,B 0.000,C 90.000,E1 31.671} C_DIS
LIN {X 0.097,Y -386.139,Z 1552.952,A 0.000,B 0.000,C 90.000,E1 27.385} C_DIS
LIN {X -0.097,Y -382.946,Z 1552.938,A 0.000,B 0.000,C 90.000,E1 24.899} C_DIS
LIN {X 0.002,Y -376.239,Z 1552.912,A 0.000,B 0.000,C 90.000,E1 20.174} C_DIS
LIN {X -0.134,Y -373.734,Z 1552.898,A 0.000,B 0.000,C 90.000,E1 17.638} C_DIS
LIN {X 0.110,Y -371.874,Z 1552.890,A 0.000,B 0.000,C 90.000,E1 16.134} C_DIS
LIN {X 0.087,Y -366.859,Z 1552.859,A 0.000,B 0.000,C 90.000,E1 10.602} C_DIS
LIN {X 0.164,Y -366.454,Z 1552.855,A 0.000,B 0.000,C 90.000,E1 9.849} C_DIS
LIN {X 0.101,Y -361.766,Z 1552.822,A 0.000,B 0.000,C 90.000,E1 3.898} C_DIS
LIN {X -0.013,Y -360.890,Z 1552.801,A 0.000,B 0.000,C 90.000,E1 0.172} C_DIS
LIN {X -0.053,Y -359.426,Z 1552.770,A 0.000,B 0.000,C 90.000,E1 354.546} C_DIS
LIN {X 0.070,Y -358.890,Z 1552.759,A 0.000,B 0.000,C 90.000,E1 352.648} C_DIS
LIN {X -0.020,Y -359.563,Z 1552.726,A 0.000,B 0.000,C 90.000,E1 346.645} C_DIS
LIN {X 0.001,Y -361.801,Z 1552.684,A 0.000,B 0.000,C 90.000,E1 339.135} C_DIS
LIN {X -0.154,Y -362.053,Z 1552.680,A 0.000,B 0.000,C 90.000,E1 338.411} C_DIS
LIN {X 0.189,Y -365.980,Z 1552.643,A 0.000,B 0.000,C 90.000,E1 331.641} C_DIS
LIN {X 0.029,Y -366.387,Z 1552.639,A 0.000,B 0.000,C 90.000,E1 330.923} C_DIS
LIN {X -0.031,Y -371.355,Z 1552.604,A 0.000,B 0.000,C 90.000,E1 324.642} C_DIS
LIN {X -0.043,Y -371.766,Z 1552.602,A 0.000,B 0.000,C 90.000,E1 324.276} C_DIS
LIN {X 0.013,Y -377.358,Z 1552.567,A 0.000,B 0.000,C 90.000,E1 318.038} C_DIS
LIN {X 0.012,Y -378.235,Z 1552.563,A 0.000,B 0.000,C 90.000,E1 317.310} C_DIS
LIN {X 0.002,Y -383.940,Z 1552.531,A 0.000,B 0.000,C 90.000,E1 311.515} C_DIS
LIN {X 0.088,Y -384.893,Z 1552.527,A 0.000,B 0.000,C 90.000,E1 310.782} C_DIS
LIN {X 0.262,Y -390.610,Z 1552.495,A 0.000,B 0.000,C 90.000,E1 305.025} C_DIS
LIN {X 0.106,Y -391.104,Z 1552.493,A 0.000,B 0.000,C 90.000,E1 304.692} C_DIS
LIN {X 0.022,Y -391.648,Z 1552.489,A 0.000,B 0.000,C 90.000,E1 303.992} C_DIS
LIN {X -0.080,Y -396.825,Z 1552.459,A 0.000,B 0.000,C 90.000,E1 298.693} C_DIS
LIN {X -0.210,Y -397.120,Z 1552.457,A 0.000,B 0.000,C 90.000,E1 298.359} C_DIS
LIN {X -0.055,Y -401.597,Z 1552.426,A 0.000,B 0.000,C 90.000,E1 292.717} C_DIS
LIN {X 0.222,Y -404.659,Z 1552.395,A 0.000,B 0.000,C 90.000,E1 287.094} C_DIS
LIN {X -0.079,Y -404.735,Z 1552.391,A 0.000,B 0.000,C 90.000,E1 286.441} C_DIS
LIN {X 0.214,Y -406.099,Z 1552.364,A 0.000,B 0.000,C 90.000,E1 281.535} C_DIS
LIN {X -0.176,Y -406.094,Z 1552.362,A 0.000,B 0.000,C 90.000,E1 281.243} C_DIS
LIN {X -0.097,Y -405.680,Z 1552.333,A 0.000,B 0.000,C 90.000,E1 276.024} C_DIS
LIN {X -0.165,Y -405.058,Z 1552.328,A 0.000,B 0.000,C 90.000,E1 274.992} C_DIS
LIN {X -0.060,Y -403.497,Z 1552.304,A 0.000,B 0.000,C 90.000,E1 270.802} C_DIS
LIN {X -0.092,Y -403.288,Z 1552.302,A 0.000,B 0.000,C 90.000,E1 270.458} C_DIS
LIN {X 0.091,Y -398.931,Z 1552.271,A 0.000,B 0.000,C 90.000,E1 264.837} C_DIS
LIN {X -0.040,Y -393.108,Z 1552.242,A 0.000,B 0.000,C 90.000,E1 259.567} C_DIS
LIN {X -0.079,Y -392.835,Z 1552.240,A 0.000,B 0.000,C 90.000,E1 259.218} C_DIS
LIN {X 0.034,Y -385.993,Z 1552.212,A 0.000,B 0.000,C 90.000,E1 254.212} C_DIS
LIN {X -0.026,Y -385.267,Z 1552.208,A 0.000,B 0.000,C 90.000,E1 253.504} C_DIS
LIN {X -0.004,Y -384.768,Z 1552.206,A 0.000,B 0.000,C 90.000,E1 253.142} C_DIS
LIN {X 0.221,Y -377.973,Z 1552.182,A 0.000,B 0.000,C 90.000,E1 248.773} C_DIS
LIN {X -0.044,Y -376.233,Z 1552.174,A 0.000,B 0.000,C 90.000,E1 247.358} C_DIS
LIN {X 0.057,Y -374.944,Z 1552.170,A 0.000,B 0.000,C 90.000,E1 246.613} C_DIS
LIN {X -0.208,Y -368.417,Z 1552.148,A 0.000,B 0.000,C 90.000,E1 242.615} C_DIS
LIN {X 0.097,Y -366.047,Z 1552.137,A 0.000,B 0.000,C 90.000,E1 240.717} C_DIS
LIN {X 0.004,Y -359.196,Z 1552.115,A 0.000,B 0.000,C 90.000,E1 236.628} C_DIS
LIN {X 0.021,Y -355.842,Z 1552.100,A 0.000,B 0.000,C 90.000,E1 233.989} C_DIS
LIN {X -0.173,Y -348.793,Z 1552.075,A 0.000,B 0.000,C 90.000,E1 229.461} C_DIS
LIN {X -0.097,Y -346.185,Z 1552.062,A 0.000,B 0.000,C 90.000,E1 227.148} C_DIS
LIN {X -0.088,Y -345.065,Z 1552.058,A 0.000,B 0.000,C 90.000,E1 226.377} C_DIS
LIN {X 0.094,Y -338.586,Z 1552.030,A 0.000,B 0.000,C 90.000,E1 221.310} C_DIS
LIN {X 0.094,Y -336.840,Z 1552.019,A 0.000,B 0.000,C 90.000,E1 219.358} C_DIS
LIN {X 0.014,Y -330.861,Z 1551.988,A 0.000,B 0.000,C 90.000,E1 213.865} C_DIS
LIN {X 0.149,Y -329.296,Z 1551.975,A 0.000,B 0.000,C 90.000,E1 211.465} C_DIS
LIN {X -0.154,Y -324.669,Z 1551.942,A 0.000,B 0.000,C 90.000,E1 205.540} C_DIS
LIN {X 0.174,Y -323.837,Z 1551.928,A 0.000,B 0.000,C 90.000,E1 203.078} C_DIS
LIN {X -0.017,Y -321.124,Z 1551.881,A 0.000,B 0.000,C 90.000,E1 194.662} C_DIS
LIN {X 0.138,Y -320.932,Z 1551.877,A 0.000,B 0.000,C 90.000,E1 193.828} C_DIS
LIN {X -0.076,Y -321.562,Z 1551.832,A 0.000,B 0.000,C 90.000,E1 185.796} C_DIS
LIN {X -0.143,Y -324.415,Z 1551.790,A 0.000,B 0.000,C 90.000,E1 178.165} C_DIS
LIN {X -0.141,Y -325.376,Z 1551.783,A 0.000,B 0.000,C 90.000,E1 176.963} C_DIS
LIN {X -0.100,Y -329.112,Z 1551.750,A 0.000,B 0.000,C 90.000,E1 170.971} C_DIS
LIN {X 0.061,Y -334.260,Z 1551.726,A 0.000,B 0.000,C 90.000,E1 166.589} C_DIS
LIN {X 0.067,Y -335.488,Z 1551.719,A 0.000,B 0.000,C 90.000,E1 165.408} C_DIS
LIN {X 0.143,Y -340.932,Z 1551.695,A 0.000,B 0.000,C 90.000,E1 161.094} C_DIS
LIN {X -0.172,Y -342.138,Z 1551.691,A 0.000,B 0.000,C 90.000,E1 160.369} C_DIS
LIN {X -0.058,Y -347.939,Z 1551.667,A 0.000,B 0.000,C 90.000,E1 156.102} C_DIS
LIN {X -0.081,Y -354.259,Z 1551.648,A 0.000,B 0.000,C 90.000,E1 152.666} C_DIS
LIN {X -0.222,Y -361.406,Z 1551.625,A 0.000,B 0.000,C 90.000,E1 148.535} C_DIS
LIN {X 0.065,Y -368.758,Z 1551.606,A 0.000,B 0.000,C 90.000,E1 145.135} C_DIS
LIN {X 0.065,Y -377.029,Z 1551.584,A 0.000,B 0.000,C 90.000,E1 141.090} C_DIS
LIN {X -0.061,Y -383.435,Z 1551.570,A 0.000,B 0.000,C 90.000,E1 138.566} C_DIS
LIN {X -0.015,Y -385.037,Z 1551.566,A 0.000,B 0.000,C 90.000,E1 137.838} C_DIS
LIN {X -0.004,Y -394.325,Z 1551.544,A 0.000,B 0.000,C 90.000,E1 133.905} C_DIS
LIN {X 0.107,Y -399.276,Z 1551.534,A 0.000,B 0.000,C 90.000,E1 132.123} C_DIS
LIN {X 0.210,Y -400.192,Z 1551.532,A 0.000,B 0.000,C 90.000,E1 131.757} C_DIS
LIN {X -0.113,Y -409.687,Z 1551.511,A 0.000,B 0.000,C 90.000,E1 127.971} C_DIS
LIN {X 0.046,Y -415.746,Z 1551.499,A 0.000,B 0.000,C 90.000,E1 125.884} C_DIS
LIN {X -0.072,Y -422.096,Z 1551.485,A 0.000,B 0.000,C 90.000,E1 123.293} C_DIS
LIN {X -0.144,Y -547.424,Z 1551.485,A 0.000,B 0.000,C 90.000,E1 123.293} C_DIS
LIN {X 0.014,Y -548.998,Z 1551.484,A 0.000,B 0.000,C 90.000,E1 123.166} C_DIS
LIN {X -0.069,Y -550.262,Z 1551.483,A 0.000,B 0.000,C 90.000,E1 122.959} C_DIS
LIN {X -0.024,Y -551.324,Z 1551.482,A 0.000,B 0.000,C 90.000,E1 122.673} C_DIS
LIN {X -0.271,Y -552.109,Z 1551.480,A 0.000,B 0.000,C 90.000,E1 122.418} C_DIS
LIN {X 0.304,Y -553.296,Z 1551.477,A 0.000,B 0.000,C 90.000,E1 121.799} C_DIS
LIN {X -0.106,Y -554.570,Z 1551.472,A 0.000,B 0.000,C 90.000,E1 121.003} C_DIS
LIN {X 0.258,Y -555.539,Z 1551.468,A 0.000,B 0.000,C 90.000,E1 120.129} C_DIS
LIN {X 0.138,Y -556.475,Z 1551.461,A 0.000,B 0.000,C 90.000,E1 119.027} C_DIS
LIN {X 0.300,Y -557.062,Z 1551.455,A 0.000,B 0.000,C 90.000,E1 117.897} C_DIS
LIN {X -0.012,Y -557.583,Z 1551.448,A 0.000,B 0.000,C 90.000,E1 116.539} C_DIS
LIN {X 0.150,Y -558.063,Z 1551.441,A 0.000,B 0.000,C 90.000,E1 115.412} C_DIS
LIN {X -0.091,Y -558.535,Z 1551.432,A 0.000,B 0.000,C 90.000,E1 113.770} C_DIS
LIN {X 0.180,Y -558.793,Z 1551.423,A 0.000,B 0.000,C 90.000,E1 112.078} C_DIS
LIN {X 0.035,Y -559.128,Z 1551.414,A 0.000,B 0.000,C 90.000,E1 110.429} C_DIS
LIN {X 0.020,Y -559.461,Z 1551.403,A 0.000,B 0.000,C 90.000,E1 108.489} C_DIS
LIN {X -0.290,Y -559.791,Z 1551.394,A 0.000,B 0.000,C 90.000,E1 106.858} C_DIS
LIN {X -0.083,Y -560.055,Z 1551.383,A 0.000,B 0.000,C 90.000,E1 104.898} C_DIS
LIN {X -0.301,Y -560.217,Z 1551.375,A 0.000,B 0.000,C 90.000,E1 103.536} C_DIS
LIN {X 0.169,Y -560.625,Z 1551.366,A 0.000,B 0.000,C 90.000,E1 101.827} C_DIS
LIN {X -0.230,Y -561.365,Z 1551.352,A 0.000,B 0.000,C 90.000,E1 99.378} C_DIS
LIN {X -0.200,Y -561.770,Z 1551.344,A 0.000,B 0.000,C 90.000,E1 97.992} C_DIS
LIN {X 0.079,Y -562.345,Z 1551.334,A 0.000,B 0.000,C 90.000,E1 96.030} C_DIS
LIN {X 0.222,Y -562.843,Z 1551.324,A 0.000,B 0.000,C 90.000,E1 94.359} C_DIS
LIN {X 0.091,Y -563.153,Z 1551.318,A 0.000,B 0.000,C 90.000,E1 93.269} C_DIS
LIN {X -0.267,Y -563.641,Z 1551.307,A 0.000,B 0.000,C 90.000,E1 91.375} C_DIS
LIN {X 0.265,Y -564.090,Z 1551.300,A 0.000,B 0.000,C 90.000,E1 89.943} C_DIS
LIN {X 0.020,Y -564.872,Z 1551.288,A 0.000,B 0.000,C 90.000,E1 87.764} C_DIS
LIN {X 0.278,Y -565.555,Z 1551.277,A 0.000,B 0.000,C 90.000,E1 85.812} C_DIS
LIN {X 0.134,Y -566.570,Z 1551.265,A 0.000,B 0.000,C 90.000,E1 83.628} C_DIS
LIN {X -0.038,Y -567.684,Z 1551.254,A 0.000,B 0.000,C 90.000,E1 81.724} C_DIS
LIN {X -0.009,Y -569.064,Z 1551.243,A 0.000,B 0.000,C 90.000,E1 79.803} C_DIS
LIN {X 0.056,Y -570.467,Z 1551.233,A 0.000,B 0.000,C 90.000,E1 77.881} C_DIS
LIN {X 0.014,Y -571.543,Z 1551.225,A 0.000,B 0.000,C 90.000,E1 76.520} C_DIS
LIN {X -0.144,Y -572.565,Z 1551.218,A 0.000,B 0.000,C 90.000,E1 75.172} C_DIS
LIN {X -0.170,Y -573.681,Z 1551.207,A 0.000,B 0.000,C 90.000,E1 73.268} C_DIS
LIN {X -0.186,Y -574.671,Z 1551.198,A 0.000,B 0.000,C 90.000,E1 71.638} C_DIS
LIN {X -0.182,Y -575.556,Z 1551.189,A 0.000,B 0.000,C 90.000,E1 70.007} C_DIS
LIN {X -0.132,Y -576.696,Z 1551.178,A 0.000,B 0.000,C 90.000,E1 68.103} C_DIS
LIN {X 0.164,Y -577.913,Z 1551.168,A 0.000,B 0.000,C 90.000,E1 66.177} C_DIS
LIN {X 0.196,Y -579.007,Z 1551.157,A 0.000,B 0.000,C 90.000,E1 64.280} C_DIS
LIN {X 0.133,Y -580.123,Z 1551.148,A 0.000,B 0.000,C 90.000,E1 62.666} C_DIS
LIN {X 0.093,Y -580.836,Z 1551.142,A 0.000,B 0.000,C 90.000,E1 61.591} C_DIS
LIN {X -0.167,Y -581.884,Z 1551.133,A 0.000,B 0.000,C 90.000,E1 59.999} C_DIS
LIN {X -0.207,Y -583.453,Z 1551.120,A 0.000,B 0.000,C 90.000,E1 57.582} C_DIS
LIN {X -0.144,Y -584.141,Z 1551.114,A 0.000,B 0.000,C 90.000,E1 56.501} C_DIS
LIN {X 0.068,Y -584.429,Z 1551.109,A 0.000,B 0.000,C 90.000,E1 55.674} C_DIS
LIN {X -0.196,Y -584.472,Z 1551.105,A 0.000,B 0.000,C 90.000,E1 54.895} C_DIS
LIN {X 0.198,Y -583.895,Z 1551.099,A 0.000,B 0.000,C 90.000,E1 53.783} C_DIS
LIN {X -0.089,Y -583.656,Z 1551.097,A 0.000,B 0.000,C 90.000,E1 53.543} C_DIS
LIN {X -0.073,Y -582.828,Z 1551.094,A 0.000,B 0.000,C 90.000,E1 53.004} C_DIS
LIN {X 0.105,Y -582.198,Z 1551.093,A 0.000,B 0.000,C 90.000,E1 52.718} C_DIS
LIN {X -0.179,Y -581.321,Z 1551.091,A 0.000,B 0.000,C 90.000,E1 52.477} C_DIS
LIN {X 0.087,Y -580.692,Z 1551.091,A 0.000,B 0.000,C 90.000,E1 52.316} C_DIS
LIN {X -0.003,Y -579.679,Z 1551.090,A 0.000,B 0.000,C 90.000,E1 52.190} C_DIS
LIN {X 0.211,Y -578.674,Z 1551.090,A 0.000,B 0.000,C 90.000,E1 52.110} C_DIS
LIN {X 0.179,Y -578.524,Z 1551.090,A 0.000,B 0.000,C 90.000,E1 52.110} C_DIS
LIN {X 0.111,Y -433.942,Z 1551.090,A 0.000,B 0.000,C 90.000,E1 52.110} C_DIS
LIN {X -0.030,Y -431.708,Z 1551.083,A 0.000,B 0.000,C 90.000,E1 50.928} C_DIS
LIN {X -0.122,Y -430.101,Z 1551.079,A 0.000,B 0.000,C 90.000,E1 50.275} C_DIS
LIN {X 0.012,Y -420.551,Z 1551.055,A 0.000,B 0.000,C 90.000,E1 45.891} C_DIS
LIN {X -0.015,Y -418.739,Z 1551.049,A 0.000,B 0.000,C 90.000,E1 44.879} C_DIS
LIN {X -0.048,Y -409.812,Z 1551.027,A 0.000,B 0.000,C 90.000,E1 40.782} C_DIS
LIN {X -0.013,Y -406.213,Z 1551.015,A 0.000,B 0.000,C 90.000,E1 38.705} C_DIS
LIN {X -0.186,Y -405.578,Z 1551.013,A 0.000,B 0.000,C 90.000,E1 38.382} C_DIS
LIN {X -0.122,Y -396.749,Z 1550.988,A 0.000,B 0.000,C 90.000,E1 33.833} C_DIS
LIN {X 0.187,Y -393.538,Z 1550.976,A 0.000,B 0.000,C 90.000,E1 31.671} C_DIS
LIN {X -0.060,Y -386.179,Z 1550.952,A 0.000,B 0.000,C 90.000,E1 27.436} C_DIS
LIN {X 0.087,Y -382.976,Z 1550.938,A 0.000,B 0.000,C 90.000,E1 24.899} C_DIS
LIN {X 0.068,Y -376.694,Z 1550.914,A 0.000,B 0.000,C 90.000,E1 20.556} C_DIS
LIN {X 0.050,Y -373.757,Z 1550.898,A 0.000,B 0.000,C 90.000,E1 17.638} C_DIS
LIN {X -0.003,Y -372.857,Z 1550.894,A 0.000,B 0.000,C 90.000,E1 16.913} C_DIS
LIN {X -0.100,Y -367.593,Z 1550.865,A 0.000,B 0.000,C 90.000,E1 11.771} C_DIS
LIN {X -0.016,Y -366.474,Z 1550.855,A 0.000,B 0.000,C 90.000,E1 9.905} C_DIS
LIN {X -0.078,Y -361.779,Z 1550.822,A 0.000,B 0.000,C 90.000,E1 3.955} C_DIS
LIN {X 0.167,Y -360.897,Z 1550.801,A 0.000,B 0.000,C 90.000,E1 0.172} C_DIS
LIN {X -0.053,Y -359.426,Z 1550.770,A 0.000,B 0.000,C 90.000,E1 354.546} C_DIS
LIN {X 0.070,Y -358.890,Z 1550.759,A 0.000,B 0.000,C 90.000,E1 352.648} C_DIS
LIN {X -0.020,Y -359.563,Z 1550.726,A 0.000,B 0.000,C 90.000,E1 346.645} C_DIS
LIN {X 0.001,Y -361.801,Z 1550.684,A 0.000,B 0.000,C 90.000,E1 339.135} C_DIS
LIN {X -0.154,Y -362.053,Z 1550.680,A 0.000,B 0.000,C 90.000,E1 338.411} C_DIS
LIN {X 0.189,Y -365.980,Z 1550.643,A 0.000,B 0.000,C 90.000,E1 331.641} C_DIS
LIN {X 0.029,Y -366.387,Z 1550.639,A 0.000,B 0.000,C 90.000,E1 330.923} C_DIS
LIN {X -0.031,Y -371.355,Z 1550.604,A 0.000,B 0.000,C 90.000,E1 324.642} C_DIS
LIN {X -0.043,Y -371.766,Z 1550.602,A 0.000,B 0.000,C 90.000,E1 324.276} C_DIS
LIN {X 0.013,Y -377.358,Z 1550.567,A 0.000,B 0.000,C 90.000,E1 318.038} C_DIS
LIN {X 0.012,Y -378.235,Z 1550.563,A 0.000,B 0.000,C 90.000,E1 317.310} C_DIS
LIN {X 0.002,Y -383.940,Z 1550.531,A 0.000,B 0.000,C 90.000,E1 311.515} C_DIS
LIN {X 0.088,Y -384.893,Z 1550.527,A 0.000,B 0.000,C 90.000,E1 310.782} C_DIS
LIN {X 0.262,Y -390.610,Z 1550.495,A 0.000,B 0.000,C 90.000,E1 305.025} C_DIS
LIN {X 0.106,Y -391.104,Z 1550.493,A 0.000,B 0.000,C 90.000,E1 304.692} C_DIS
LIN {X 0.022,Y -391.648,Z 1550.489,A 0.000,B 0.000,C 90.000,E1 303.992} C_DIS
LIN {X -0.080,Y -396.825,Z 1550.459,A 0.000,B 0.000,C 90.000,E1 298.693} C_DIS
LIN {X -0.210,Y -397.120,Z 1550.457,A 0.000,B 0.000,C 90.000,E1 298.359} C_DIS
LIN {X -0.055,Y -401.597,Z 1550.426,A 0.000,B 0.000,C 90.000,E1 292.717} C_DIS
LIN {X 0.222,Y -404.659,Z 1550.395,A 0.000,B 0.000,C 90.000,E1 287.094} C_DIS
LIN {X -0.079,Y -404.735,Z 1550.391,A 0.000,B 0.000,C 90.000,E1 286.441} C_DIS
LIN {X 0.214,Y -406.099,Z 1550.364,A 0.000,B 0.000,C 90.000,E1 281.535} C_DIS
LIN {X -0.176,Y -406.094,Z 1550.362,A 0.000,B 0.000,C 90.000,E1 281.243} C_DIS
LIN {X -0.097,Y -405.680,Z 1550.333,A 0.000,B 0.000,C 90.000,E1 276.024} C_DIS
LIN {X -0.165,Y -405.058,Z 1550.328,A 0.000,B 0.000,C 90.000,E1 274.992} C_DIS
LIN {X -0.060,Y -403.497,Z 1550.304,A 0.000,B 0.000,C 90.000,E1 270.802} C_DIS
LIN {X -0.092,Y -403.288,Z 1550.302,A 0.000,B 0.000,C 90.000,E1 270.458} C_DIS
LIN {X 0.091,Y -398.931,Z 1550.271,A 0.000,B 0.000,C 90.000,E1 264.837} C_DIS
LIN {X -0.040,Y -393.108,Z 1550.242,A 0.000,B 0.000,C 90.000,E1 259.567} C_DIS
LIN {X -0.079,Y -392.835,Z 1550.240,A 0.000,B 0.000,C 90.000,E1 259.218} C_DIS
LIN {X 0.034,Y -385.993,Z 1550.212,A 0.000,B 0.000,C 90.000,E1 254.212} C_DIS
LIN {X -0.026,Y -385.267,Z 1550.208,A 0.000,B 0.000,C 90.000,E1 253.504} C_DIS
LIN {X -0.004,Y -384.768,Z 1550.206,A 0.000,B 0.000,C 90.000,E1 253.142} C_DIS
LIN {X 0.221,Y -377.973,Z 1550.182,A 0.000,B 0.000,C 90.000,E1 248.773} C_DIS
LIN {X -0.044,Y -376.233,Z 1550.174,A 0.000,B 0.000,C 90.000,E1 247.358} C_DIS
LIN {X 0.057,Y -374.944,Z 1550.170,A 0.000,B 0.000,C 90.000,E1 246.613} C_DIS
LIN {X -0.208,Y -368.417,Z 1550.148,A 0.000,B 0.000,C 90.000,E1 242.615} C_DIS
LIN {X 0.097,Y -366.047,Z 1550.137,A 0.000,B 0.000,C 90.000,E1 240.717} C_DIS
LIN {X 0.004,Y -359.196,Z 1550.115,A 0.000,B 0.000,C 90.000,E1 236.628} C_DIS
LIN {X 0.021,Y -355.842,Z 1550.100,A 0.000,B 0.000,C 90.000,E1 233.989} C_DIS
LIN {X -0.173,Y -348.793,Z 1550.075,A 0.000,B 0.000,C 90.000,E1 229.461} C_DIS
LIN {X -0.097,Y -346.185,Z 1550.062,A 0.000,B 0.000,C 90.000,E1 227.148} C_DIS
LIN {X -0.088,Y -345.065,Z 1550.058,A 0.000,B 0.000,C 90.000,E1 226.377} C_DIS
LIN {X 0.094,Y -338.586,Z 1550.030,A 0.000,B 0.000,C 90.000,E1 221.310} C_DIS
LIN {X 0.094,Y -336.840,Z 1550.019,A 0.000,B 0.000,C 90.000,E1 219.358} C_DIS
LIN {X 0.014,Y -330.861,Z 1549.988,A 0.000,B 0.000,C 90.000,E1 213.865} C_DIS
LIN {X 0.149,Y -329.296,Z 1549.975,A 0.000,B 0.000,C 90.000,E1 211.465} C_DIS
LIN {X -0.154,Y -324.669,Z 1549.942,A 0.000,B 0.000,C 90.000,E1 205.540} C_DIS
LIN {X 0.174,Y -323.837,Z 1549.928,A 0.000,B 0.000,C 90.000,E1 203.078} C_DIS
LIN {X -0.017,Y -321.124,Z 1549.881,A 0.000,B 0.000,C 90.000,E1 194.662} C_DIS
LIN {X 0.138,Y -320.932,Z 1549.877,A 0.000,B 0.000,C 90.000,E1 193.828} C_DIS
LIN {X -0.076,Y -321.562,Z 1549.832,A 0.000,B 0.000,C 90.000,E1 185.796} C_DIS
LIN {X -0.143,Y -324.415,Z 1549.790,A 0.000,B 0.000,C 90.000,E1 178.165} C_DIS
LIN {X -0.141,Y -325.376,Z 1549.783,A 0.000,B 0.000,C 90.000,E1 176.963} C_DIS
LIN {X -0.100,Y -329.112,Z 1549.750,A 0.000,B 0.000,C 90.000,E1 170.971} C_DIS
LIN {X 0.061,Y -334.260,Z 1549.726,A 0.000,B 0.000,C 90.000,E1 166.589} C_DIS
LIN {X 0.067,Y -335.488,Z 1549.719,A 0.000,B 0.000,C 90.000,E1 165.408} C_DIS
LIN {X 0.143,Y -340.932,Z 1549.695,A 0.000,B 0.000,C 90.000,E1 161.094} C_DIS
LIN {X -0.172,Y -342.138,Z 1549.691,A 0.000,B 0.000,C 90.000,E1 160.369} C_DIS
LIN {X -0.058,Y -347.939,Z 1549.667,A 0.000,B 0.000,C 90.000,E1 156.102} C_DIS
LIN {X -0.081,Y -354.259,Z 1549.648,A 0.000,B 0.000,C 90.000,E1 152.666} C_DIS
LIN {X -0.222,Y -361.406,Z 1549.625,A 0.000,B 0.000,C 90.000,E1 148.535} C_DIS
LIN {X 0.065,Y -368.758,Z 1549.606,A 0.000,B 0.000,C 90.000,E1 145.135} C_DIS
LIN {X 0.065,Y -377.029,Z 1549.584,A 0.000,B 0.000,C 90.000,E1 141.090} C_DIS
LIN {X -0.061,Y -383.435,Z 1549.570,A 0.000,B 0.000,C 90.000,E1 138.566} C_DIS
LIN {X -0.015,Y -385.037,Z 1549.566,A 0.000,B 0.000,C 90.000,E1 137.838} C_DIS
LIN {X -0.004,Y -394.325,Z 1549.544,A 0.000,B 0.000,C 90.000,E1 133.905} C_DIS
LIN {X 0.107,Y -399.276,Z 1549.534,A 0.000,B 0.000,C 90.000,E1 132.123} C_DIS
LIN {X 0.210,Y -400.192,Z 1549.532,A 0.000,B 0.000,C 90.000,E1 131.757} C_DIS
LIN {X -0.113,Y -409.687,Z 1549.511,A 0.000,B 0.000,C 90.000,E1 127.971} C_DIS
LIN {X 0.046,Y -415.746,Z 1549.499,A 0.000,B 0.000,C 90.000,E1 125.884} C_DIS
LIN {X -0.048,Y -419.052,Z 1549.492,A 0.000,B 0.000,C 90.000,E1 124.485} C_DIS
LIN {X -0.112,Y -547.100,Z 1549.492,A 0.000,B 0.000,C 90.000,E1 124.485} C_DIS
LIN {X 0.026,Y -547.809,Z 1549.491,A 0.000,B 0.000,C 90.000,E1 124.452} C_DIS
LIN {X -0.053,Y -549.272,Z 1549.491,A 0.000,B 0.000,C 90.000,E1 124.326} C_DIS
LIN {X -0.131,Y -550.076,Z 1549.490,A 0.000,B 0.000,C 90.000,E1 124.199} C_DIS
LIN {X -0.081,Y -551.249,Z 1549.488,A 0.000,B 0.000,C 90.000,E1 123.913} C_DIS
LIN {X -0.030,Y -552.117,Z 1549.487,A 0.000,B 0.000,C 90.000,E1 123.627} C_DIS
LIN {X -0.221,Y -553.378,Z 1549.484,A 0.000,B 0.000,C 90.000,E1 123.086} C_DIS
LIN {X 0.067,Y -554.256,Z 1549.481,A 0.000,B 0.000,C 90.000,E1 122.498} C_DIS
LIN {X -0.039,Y -555.206,Z 1549.476,A 0.000,B 0.000,C 90.000,E1 121.671} C_DIS
LIN {X 0.112,Y -556.112,Z 1549.470,A 0.000,B 0.000,C 90.000,E1 120.541} C_DIS
LIN {X -0.209,Y -556.738,Z 1549.464,A 0.000,B 0.000,C 90.000,E1 119.461} C_DIS
LIN {X 0.228,Y -557.325,Z 1549.456,A 0.000,B 0.000,C 90.000,E1 118.025} C_DIS
LIN {X -0.080,Y -557.809,Z 1549.448,A 0.000,B 0.000,C 90.000,E1 116.668} C_DIS
LIN {X -0.125,Y -558.349,Z 1549.440,A 0.000,B 0.000,C 90.000,E1 115.283} C_DIS
LIN {X 0.152,Y -558.806,Z 1549.431,A 0.000,B 0.000,C 90.000,E1 113.590} C_DIS
LIN {X -0.088,Y -559.072,Z 1549.422,A 0.000,B 0.000,C 90.000,E1 111.950} C_DIS
LIN {X -0.230,Y -559.361,Z 1549.413,A 0.000,B 0.000,C 90.000,E1 110.301} C_DIS
LIN {X 0.163,Y -559.655,Z 1549.403,A 0.000,B 0.000,C 90.000,E1 108.598} C_DIS
LIN {X 0.085,Y -559.955,Z 1549.396,A 0.000,B 0.000,C 90.000,E1 107.221} C_DIS
LIN {X 0.156,Y -560.159,Z 1549.387,A 0.000,B 0.000,C 90.000,E1 105.552} C_DIS
LIN {X 0.079,Y -560.382,Z 1549.379,A 0.000,B 0.000,C 90.000,E1 104.175} C_DIS
LIN {X 0.180,Y -560.832,Z 1549.367,A 0.000,B 0.000,C 90.000,E1 101.951} C_DIS
LIN {X -0.045,Y -561.652,Z 1549.351,A 0.000,B 0.000,C 90.000,E1 99.208} C_DIS
LIN {X -0.077,Y -561.999,Z 1549.345,A 0.000,B 0.000,C 90.000,E1 98.106} C_DIS
LIN {X 0.203,Y -562.590,Z 1549.334,A 0.000,B 0.000,C 90.000,E1 96.144} C_DIS
LIN {X 0.254,Y -563.013,Z 1549.327,A 0.000,B 0.000,C 90.000,E1 94.759} C_DIS
LIN {X -0.211,Y -563.478,Z 1549.317,A 0.000,B 0.000,C 90.000,E1 93.151} C_DIS
LIN {X -0.028,Y -563.971,Z 1549.307,A 0.000,B 0.000,C 90.000,E1 91.203} C_DIS
LIN {X -0.053,Y -564.446,Z 1549.299,A 0.000,B 0.000,C 90.000,E1 89.828} C_DIS
LIN {X 0.277,Y -565.281,Z 1549.287,A 0.000,B 0.000,C 90.000,E1 87.593} C_DIS
LIN {X -0.023,Y -565.996,Z 1549.276,A 0.000,B 0.000,C 90.000,E1 85.698} C_DIS
LIN {X -0.161,Y -566.991,Z 1549.264,A 0.000,B 0.000,C 90.000,E1 83.514} C_DIS
LIN {X -0.244,Y -568.163,Z 1549.253,A 0.000,B 0.000,C 90.000,E1 81.602} C_DIS
LIN {X -0.293,Y -569.572,Z 1549.243,A 0.000,B 0.000,C 90.000,E1 79.690} C_DIS
LIN {X -0.102,Y -571.000,Z 1549.232,A 0.000,B 0.000,C 90.000,E1 77.757} C_DIS
LIN {X -0.072,Y -572.312,Z 1549.223,A 0.000,B 0.000,C 90.000,E1 76.117} C_DIS
LIN {X -0.271,Y -573.063,Z 1549.217,A 0.000,B 0.000,C 90.000,E1 75.046} C_DIS
LIN {X -0.277,Y -574.213,Z 1549.206,A 0.000,B 0.000,C 90.000,E1 73.142} C_DIS
LIN {X 0.269,Y -575.200,Z 1549.197,A 0.000,B 0.000,C 90.000,E1 71.456} C_DIS
LIN {X 0.117,Y -576.217,Z 1549.187,A 0.000,B 0.000,C 90.000,E1 69.571} C_DIS
LIN {X -0.189,Y -577.247,Z 1549.178,A 0.000,B 0.000,C 90.000,E1 67.975} C_DIS
LIN {X -0.025,Y -578.558,Z 1549.166,A 0.000,B 0.000,C 90.000,E1 65.793} C_DIS
LIN {X -0.113,Y -579.857,Z 1549.154,A 0.000,B 0.000,C 90.000,E1 63.640} C_DIS
LIN {X -0.021,Y -580.822,Z 1549.146,A 0.000,B 0.000,C 90.000,E1 62.281} C_DIS
LIN {X -0.049,Y -581.859,Z 1549.137,A 0.000,B 0.000,C 90.000,E1 60.667} C_DIS
LIN {X -0.013,Y -582.536,Z 1549.131,A 0.000,B 0.000,C 90.000,E1 59.587} C_DIS
LIN {X -0.059,Y -583.800,Z 1549.121,A 0.000,B 0.000,C 90.000,E1 57.709} C_DIS
LIN {X -0.130,Y -584.678,Z 1549.113,A 0.000,B 0.000,C 90.000,E1 56.373} C_DIS
LIN {X -0.026,Y -585.384,Z 1549.106,A 0.000,B 0.000,C 90.000,E1 55.022} C_DIS
LIN {X 0.387,Y -585.439,Z 1549.100,A 0.000,B 0.000,C 90.000,E1 53.909} C_DIS
LIN {X -0.054,Y -585.324,Z 1549.097,A 0.000,B 0.000,C 90.000,E1 53.417} C_DIS
LIN {X 0.322,Y -584.990,Z 1549.094,A 0.000,B 0.000,C 90.000,E1 52.844} C_DIS
LIN {X -0.123,Y -584.420,Z 1549.091,A 0.000,B 0.000,C 90.000,E1 52.351} C_DIS
LIN {X -0.216,Y -583.508,Z 1549.088,A 0.000,B 0.000,C 90.000,E1 51.823} C_DIS
LIN {X -0.033,Y -582.875,Z 1549.086,A 0.000,B 0.000,C 90.000,E1 51.537} C_DIS
LIN {X 0.146,Y -581.912,Z 1549.085,A 0.000,B 0.000,C 90.000,E1 51.251} C_DIS
LIN {X 0.052,Y -581.151,Z 1549.084,A 0.000,B 0.000,C 90.000,E1 51.126} C_DIS
LIN {X -0.129,Y -579.470,Z 1549.083,A 0.000,B 0.000,C 90.000,E1 51.009} C_DIS
LIN {X -0.161,Y -579.294,Z 1549.083,A 0.000,B 0.000,C 90.000,E1 51.009} C_DIS
LIN {X -0.144,Y -431.823,Z 1549.083,A 0.000,B 0.000,C 90.000,E1 51.009} C_DIS
LIN {X -0.274,Y -431.403,Z 1549.082,A 0.000,B 0.000,C 90.000,E1 50.803} C_DIS
LIN {X 0.232,Y -421.528,Z 1549.058,A 0.000,B 0.000,C 90.000,E1 46.377} C_DIS
LIN {X -0.007,Y -418.394,Z 1549.048,A 0.000,B 0.000,C 90.000,E1 44.717} C_DIS
LIN {X 0.098,Y -408.873,Z 1549.024,A 0.000,B 0.000,C 90.000,E1 40.253} C_DIS
LIN {X -0.035,Y -405.954,Z 1549.014,A 0.000,B 0.000,C 90.000,E1 38.543} C_DIS
LIN {X 0.183,Y -397.639,Z 1548.991,A 0.000,B 0.000,C 90.000,E1 34.326} C_DIS
LIN {X 0.047,Y -393.865,Z 1548.977,A 0.000,B 0.000,C 90.000,E1 31.878} C_DIS
LIN {X -0.175,Y -386.451,Z 1548.953,A 0.000,B 0.000,C 90.000,E1 27.641} C_DIS
LIN {X -0.197,Y -382.757,Z 1548.938,A 0.000,B 0.000,C 90.000,E1 24.771} C_DIS
LIN {X -0.113,Y -376.075,Z 1548.911,A 0.000,B 0.000,C 90.000,E1 20.047} C_DIS
LIN {X 0.100,Y -373.610,Z 1548.897,A 0.000,B 0.000,C 90.000,E1 17.457} C_DIS
LIN {X 0.133,Y -368.013,Z 1548.869,A 0.000,B 0.000,C 90.000,E1 12.299} C_DIS
LIN {X 0.150,Y -366.575,Z 1548.856,A 0.000,B 0.000,C 90.000,E1 10.074} C_DIS
LIN {X 0.006,Y -366.303,Z 1548.854,A 0.000,B 0.000,C 90.000,E1 9.726} C_DIS
LIN {X -0.115,Y -361.702,Z 1548.821,A 0.000,B 0.000,C 90.000,E1 3.784} C_DIS
LIN {X -0.034,Y -360.909,Z 1548.802,A 0.000,B 0.000,C 90.000,E1 0.401} C_DIS
LIN {X 0.137,Y -360.684,Z 1548.799,A 0.000,B 0.000,C 90.000,E1 359.771} C_DIS
LIN {X -0.053,Y -359.426,Z 1548.770,A 0.000,B 0.000,C 90.000,E1 354.546} C_DIS
LIN {X 0.070,Y -358.890,Z 1548.759,A 0.000,B 0.000,C 90.000,E1 352.648} C_DIS
LIN {X -0.020,Y -359.563,Z 1548.726,A 0.000,B 0.000,C 90.000,E1 346.645} C_DIS
LIN {X 0.001,Y -361.801,Z 1548.684,A 0.000,B 0.000,C 90.000,E1 339.135} C_DIS
LIN {X -0.154,Y -362.053,Z 1548.680,A 0.000,B 0.000,C 90.000,E1 338.411} C_DIS
LIN {X 0.189,Y -365.980,Z 1548.643,A 0.000,B 0.000,C 90.000,E1 331.641} C_DIS
LIN {X 0.029,Y -366.387,Z 1548.639,A 0.000,B 0.000,C 90.000,E1 330.923} C_DIS
LIN {X -0.031,Y -371.355,Z 1548.604,A 0.000,B 0.000,C 90.000,E1 324.642} C_DIS
LIN {X -0.043,Y -371.766,Z 1548.602,A 0.000,B 0.000,C 90.000,E1 324.276} C_DIS
LIN {X 0.013,Y -377.358,Z 1548.567,A 0.000,B 0.000,C 90.000,E1 318.038} C_DIS
LIN {X 0.012,Y -378.235,Z 1548.563,A 0.000,B 0.000,C 90.000,E1 317.310} C_DIS
LIN {X 0.002,Y -383.940,Z 1548.531,A 0.000,B 0.000,C 90.000,E1 311.515} C_DIS
LIN {X 0.088,Y -384.893,Z 1548.527,A 0.000,B 0.000,C 90.000,E1 310.782} C_DIS
LIN {X 0.262,Y -390.610,Z 1548.495,A 0.000,B 0.000,C 90.000,E1 305.025} C_DIS
LIN {X 0.106,Y -391.104,Z 1548.493,A 0.000,B 0.000,C 90.000,E1 304.692} C_DIS
LIN {X 0.022,Y -391.648,Z 1548.489,A 0.000,B 0.000,C 90.000,E1 303.992} C_DIS
LIN {X -0.080,Y -396.825,Z 1548.459,A 0.000,B 0.000,C 90.000,E1 298.693} C_DIS
LIN {X -0.210,Y -397.120,Z 1548.457,A 0.000,B 0.000,C 90.000,E1 298.359} C_DIS
LIN {X -0.055,Y -401.597,Z 1548.426,A 0.000,B 0.000,C 90.000,E1 292.717} C_DIS
LIN {X 0.222,Y -404.659,Z 1548.395,A 0.000,B 0.000,C 90.000,E1 287.094} C_DIS
LIN {X -0.079,Y -404.735,Z 1548.391,A 0.000,B 0.000,C 90.000,E1 286.441} C_DIS
LIN {X 0.214,Y -406.099,Z 1548.364,A 0.000,B 0.000,C 90.000,E1 281.535} C_DIS
LIN {X -0.176,Y -406.094,Z 1548.362,A 0.000,B 0.000,C 90.000,E1 281.243} C_DIS
LIN {X -0.097,Y -405.680,Z 1548.333,A 0.000,B 0.000,C 90.000,E1 276.024} C_DIS
LIN {X -0.165,Y -405.058,Z 1548.328,A 0.000,B 0.000,C 90.000,E1 274.992} C_DIS
LIN {X -0.060,Y -403.497,Z 1548.304,A 0.000,B 0.000,C 90.000,E1 270.802} C_DIS
LIN {X -0.092,Y -403.288,Z 1548.302,A 0.000,B 0.000,C 90.000,E1 270.458} C_DIS
LIN {X 0.091,Y -398.931,Z 1548.271,A 0.000,B 0.000,C 90.000,E1 264.837} C_DIS
LIN {X -0.040,Y -393.108,Z 1548.242,A 0.000,B 0.000,C 90.000,E1 259.567} C_DIS
LIN {X -0.079,Y -392.835,Z 1548.240,A 0.000,B 0.000,C 90.000,E1 259.218} C_DIS
LIN {X 0.034,Y -385.993,Z 1548.212,A 0.000,B 0.000,C 90.000,E1 254.212} C_DIS
LIN {X -0.026,Y -385.267,Z 1548.208,A 0.000,B 0.000,C 90.000,E1 253.504} C_DIS
LIN {X -0.004,Y -384.768,Z 1548.206,A 0.000,B 0.000,C 90.000,E1 253.142} C_DIS
LIN {X 0.221,Y -377.973,Z 1548.182,A 0.000,B 0.000,C 90.000,E1 248.773} C_DIS
LIN {X -0.044,Y -376.233,Z 1548.174,A 0.000,B 0.000,C 90.000,E1 247.358} C_DIS
LIN {X 0.057,Y -374.944,Z 1548.170,A 0.000,B 0.000,C 90.000,E1 246.613} C_DIS
LIN {X -0.208,Y -368.417,Z 1548.148,A 0.000,B 0.000,C 90.000,E1 242.615} C_DIS
LIN {X 0.097,Y -366.047,Z 1548.137,A 0.000,B 0.000,C 90.000,E1 240.717} C_DIS
LIN {X 0.004,Y -359.196,Z 1548.115,A 0.000,B 0.000,C 90.000,E1 236.628} C_DIS
LIN {X 0.021,Y -355.842,Z 1548.100,A 0.000,B 0.000,C 90.000,E1 233.989} C_DIS
LIN {X -0.173,Y -348.793,Z 1548.075,A 0.000,B 0.000,C 90.000,E1 229.461} C_DIS
LIN {X -0.097,Y -346.185,Z 1548.062,A 0.000,B 0.000,C 90.000,E1 227.148} C_DIS
LIN {X -0.088,Y -345.065,Z 1548.058,A 0.000,B 0.000,C 90.000,E1 226.377} C_DIS
LIN {X 0.094,Y -338.586,Z 1548.030,A 0.000,B 0.000,C 90.000,E1 221.310} C_DIS
LIN {X 0.094,Y -336.840,Z 1548.019,A 0.000,B 0.000,C 90.000,E1 219.358} C_DIS
LIN {X 0.014,Y -330.861,Z 1547.988,A 0.000,B 0.000,C 90.000,E1 213.865} C_DIS
LIN {X 0.149,Y -329.296,Z 1547.975,A 0.000,B 0.000,C 90.000,E1 211.465} C_DIS
LIN {X -0.154,Y -324.669,Z 1547.942,A 0.000,B 0.000,C 90.000,E1 205.540} C_DIS
LIN {X 0.174,Y -323.837,Z 1547.928,A 0.000,B 0.000,C 90.000,E1 203.078} C_DIS
LIN {X -0.017,Y -321.124,Z 1547.881,A 0.000,B 0.000,C 90.000,E1 194.662} C_DIS
LIN {X 0.138,Y -320.932,Z 1547.877,A 0.000,B 0.000,C 90.000,E1 193.828} C_DIS
LIN {X -0.076,Y -321.562,Z 1547.832,A 0.000,B 0.000,C 90.000,E1 185.796} C_DIS
LIN {X -0.143,Y -324.415,Z 1547.790,A 0.000,B 0.000,C 90.000,E1 178.165} C_DIS
LIN {X -0.141,Y -325.376,Z 1547.783,A 0.000,B 0.000,C 90.000,E1 176.963} C_DIS
LIN {X -0.100,Y -329.112,Z 1547.750,A 0.000,B 0.000,C 90.000,E1 170.971} C_DIS
LIN {X 0.061,Y -334.260,Z 1547.726,A 0.000,B 0.000,C 90.000,E1 166.589} C_DIS
LIN {X 0.067,Y -335.488,Z 1547.719,A 0.000,B 0.000,C 90.000,E1 165.408} C_DIS
LIN {X 0.143,Y -340.932,Z 1547.695,A 0.000,B 0.000,C 90.000,E1 161.094} C_DIS
LIN {X -0.172,Y -342.138,Z 1547.691,A 0.000,B 0.000,C 90.000,E1 160.369} C_DIS
LIN {X -0.058,Y -347.939,Z 1547.667,A 0.000,B 0.000,C 90.000,E1 156.102} C_DIS
LIN {X -0.081,Y -354.259,Z 1547.648,A 0.000,B 0.000,C 90.000,E1 152.666} C_DIS
LIN {X -0.222,Y -361.406,Z 1547.625,A 0.000,B 0.000,C 90.000,E1 148.535} C_DIS
LIN {X 0.065,Y -368.758,Z 1547.606,A 0.000,B 0.000,C 90.000,E1 145.135} C_DIS
LIN {X 0.065,Y -377.029,Z 1547.584,A 0.000,B 0.000,C 90.000,E1 141.090} C_DIS
LIN {X -0.061,Y -383.435,Z 1547.570,A 0.000,B 0.000,C 90.000,E1 138.566} C_DIS
LIN {X -0.015,Y -385.037,Z 1547.566,A 0.000,B 0.000,C 90.000,E1 137.838} C_DIS
LIN {X -0.004,Y -394.325,Z 1547.544,A 0.000,B 0.000,C 90.000,E1 133.905} C_DIS
LIN {X 0.107,Y -399.276,Z 1547.534,A 0.000,B 0.000,C 90.000,E1 132.123} C_DIS
LIN {X 0.210,Y -400.192,Z 1547.532,A 0.000,B 0.000,C 90.000,E1 131.757} C_DIS
LIN {X -0.113,Y -409.687,Z 1547.511,A 0.000,B 0.000,C 90.000,E1 127.971} C_DIS
LIN {X -0.051,Y -415.852,Z 1547.499,A 0.000,B 0.000,C 90.000,E1 125.851} C_DIS
LIN {X 0.099,Y -416.376,Z 1547.498,A 0.000,B 0.000,C 90.000,E1 125.598} C_DIS
LIN {X 0.083,Y -546.909,Z 1547.498,A 0.000,B 0.000,C 90.000,E1 125.598} C_DIS
LIN {X 0.293,Y -548.178,Z 1547.498,A 0.000,B 0.000,C 90.000,E1 125.518} C_DIS
LIN {X 0.028,Y -549.473,Z 1547.497,A 0.000,B 0.000,C 90.000,E1 125.391} C_DIS
LIN {X 0.078,Y -550.878,Z 1547.495,A 0.000,B 0.000,C 90.000,E1 125.105} C_DIS
LIN {X 0.133,Y -551.861,Z 1547.494,A 0.000,B 0.000,C 90.000,E1 124.818} C_DIS
LIN {X -0.061,Y -553.283,Z 1547.490,A 0.000,B 0.000,C 90.000,E1 124.278} C_DIS
LIN {X 0.068,Y -554.267,Z 1547.487,A 0.000,B 0.000,C 90.000,E1 123.706} C_DIS
LIN {X -0.107,Y -555.005,Z 1547.484,A 0.000,B 0.000,C 90.000,E1 123.166} C_DIS
LIN {X -0.205,Y -555.743,Z 1547.480,A 0.000,B 0.000,C 90.000,E1 122.339} C_DIS
LIN {X -0.050,Y -556.353,Z 1547.473,A 0.000,B 0.000,C 90.000,E1 121.209} C_DIS
LIN {X -0.037,Y -556.994,Z 1547.464,A 0.000,B 0.000,C 90.000,E1 119.539} C_DIS
LIN {X -0.082,Y -557.598,Z 1547.456,A 0.000,B 0.000,C 90.000,E1 118.153} C_DIS
LIN {X -0.097,Y -558.132,Z 1547.447,A 0.000,B 0.000,C 90.000,E1 116.488} C_DIS
LIN {X 0.317,Y -558.587,Z 1547.441,A 0.000,B 0.000,C 90.000,E1 115.335} C_DIS
LIN {X 0.080,Y -559.030,Z 1547.432,A 0.000,B 0.000,C 90.000,E1 113.695} C_DIS
LIN {X -0.163,Y -559.265,Z 1547.424,A 0.000,B 0.000,C 90.000,E1 112.333} C_DIS
LIN {X 0.013,Y -559.539,Z 1547.413,A 0.000,B 0.000,C 90.000,E1 110.375} C_DIS
LIN {X 0.298,Y -559.814,Z 1547.406,A 0.000,B 0.000,C 90.000,E1 108.960} C_DIS
LIN {X -0.014,Y -560.145,Z 1547.396,A 0.000,B 0.000,C 90.000,E1 107.330} C_DIS
LIN {X 0.052,Y -560.367,Z 1547.387,A 0.000,B 0.000,C 90.000,E1 105.662} C_DIS
LIN {X -0.017,Y -560.630,Z 1547.378,A 0.000,B 0.000,C 90.000,E1 104.008} C_DIS
LIN {X 0.220,Y -561.103,Z 1547.366,A 0.000,B 0.000,C 90.000,E1 101.771} C_DIS
LIN {X -0.159,Y -561.859,Z 1547.352,A 0.000,B 0.000,C 90.000,E1 99.321} C_DIS
LIN {X -0.118,Y -562.279,Z 1547.344,A 0.000,B 0.000,C 90.000,E1 97.936} C_DIS
LIN {X 0.090,Y -562.828,Z 1547.335,A 0.000,B 0.000,C 90.000,E1 96.258} C_DIS
LIN {X 0.094,Y -563.279,Z 1547.327,A 0.000,B 0.000,C 90.000,E1 94.878} C_DIS
LIN {X 0.211,Y -563.758,Z 1547.318,A 0.000,B 0.000,C 90.000,E1 93.212} C_DIS
LIN {X -0.132,Y -564.226,Z 1547.307,A 0.000,B 0.000,C 90.000,E1 91.318} C_DIS
LIN {X -0.152,Y -564.743,Z 1547.300,A 0.000,B 0.000,C 90.000,E1 89.943} C_DIS
LIN {X -0.165,Y -565.224,Z 1547.292,A 0.000,B 0.000,C 90.000,E1 88.568} C_DIS
LIN {X -0.268,Y -565.684,Z 1547.286,A 0.000,B 0.000,C 90.000,E1 87.478} C_DIS
LIN {X -0.104,Y -566.370,Z 1547.277,A 0.000,B 0.000,C 90.000,E1 85.812} C_DIS
LIN {X -0.228,Y -567.293,Z 1547.265,A 0.000,B 0.000,C 90.000,E1 83.628} C_DIS
LIN {X -0.207,Y -568.660,Z 1547.252,A 0.000,B 0.000,C 90.000,E1 81.432} C_DIS
LIN {X -0.149,Y -570.091,Z 1547.242,A 0.000,B 0.000,C 90.000,E1 79.511} C_DIS
LIN {X -0.249,Y -571.319,Z 1547.233,A 0.000,B 0.000,C 90.000,E1 77.881} C_DIS
LIN {X 0.109,Y -572.883,Z 1547.222,A 0.000,B 0.000,C 90.000,E1 75.936} C_DIS
LIN {X 0.114,Y -573.741,Z 1547.214,A 0.000,B 0.000,C 90.000,E1 74.574} C_DIS
LIN {X 0.119,Y -574.950,Z 1547.204,A 0.000,B 0.000,C 90.000,E1 72.670} C_DIS
LIN {X -0.056,Y -575.703,Z 1547.196,A 0.000,B 0.000,C 90.000,E1 71.329} C_DIS
LIN {X -0.027,Y -576.606,Z 1547.187,A 0.000,B 0.000,C 90.000,E1 69.699} C_DIS
LIN {X 0.051,Y -577.813,Z 1547.177,A 0.000,B 0.000,C 90.000,E1 67.794} C_DIS
LIN {X -0.157,Y -578.919,Z 1547.166,A 0.000,B 0.000,C 90.000,E1 65.921} C_DIS
LIN {X -0.238,Y -580.186,Z 1547.154,A 0.000,B 0.000,C 90.000,E1 63.768} C_DIS
LIN {X 0.238,Y -581.352,Z 1547.145,A 0.000,B 0.000,C 90.000,E1 62.103} C_DIS
LIN {X -0.278,Y -582.748,Z 1547.133,A 0.000,B 0.000,C 90.000,E1 59.999} C_DIS
LIN {X 0.170,Y -583.981,Z 1547.123,A 0.000,B 0.000,C 90.000,E1 58.074} C_DIS
LIN {X -0.214,Y -585.050,Z 1547.114,A 0.000,B 0.000,C 90.000,E1 56.501} C_DIS
LIN {X 0.046,Y -585.850,Z 1547.106,A 0.000,B 0.000,C 90.000,E1 55.135} C_DIS
LIN {X -0.110,Y -586.373,Z 1547.097,A 0.000,B 0.000,C 90.000,E1 53.543} C_DIS
LIN {X 0.115,Y -586.304,Z 1547.093,A 0.000,B 0.000,C 90.000,E1 52.718} C_DIS
LIN {X 0.223,Y -585.914,Z 1547.089,A 0.000,B 0.000,C 90.000,E1 51.904} C_DIS
LIN {X 0.144,Y -585.481,Z 1547.086,A 0.000,B 0.000,C 90.000,E1 51.376} C_DIS
LIN {X -0.304,Y -584.682,Z 1547.083,A 0.000,B 0.000,C 90.000,E1 50.884} C_DIS
LIN {X -0.119,Y -584.119,Z 1547.081,A 0.000,B 0.000,C 90.000,E1 50.598} C_DIS
LIN {X 0.061,Y -583.340,Z 1547.080,A 0.000,B 0.000,C 90.000,E1 50.312} C_DIS
LIN {X -0.112,Y -582.801,Z 1547.079,A 0.000,B 0.000,C 90.000,E1 50.194} C_DIS
LIN {X 0.307,Y -581.869,Z 1547.078,A 0.000,B 0.000,C 90.000,E1 49.989} C_DIS
LIN {X 0.331,Y -581.135,Z 1547.078,A 0.000,B 0.000,C 90.000,E1 49.908} C_DIS
LIN {X -0.128,Y -580.214,Z 1547.077,A 0.000,B 0.000,C 90.000,E1 49.908} C_DIS
LIN {X -0.124,Y -429.182,Z 1547.077,A 0.000,B 0.000,C 90.000,E1 49.908} C_DIS
LIN {X 0.118,Y -420.278,Z 1547.054,A 0.000,B 0.000,C 90.000,E1 45.729} C_DIS
LIN {X -0.208,Y -418.426,Z 1547.049,A 0.000,B 0.000,C 90.000,E1 44.757} C_DIS
LIN {X -0.121,Y -408.897,Z 1547.024,A 0.000,B 0.000,C 90.000,E1 40.297} C_DIS
LIN {X 0.059,Y -405.975,Z 1547.014,A 0.000,B 0.000,C 90.000,E1 38.543} C_DIS
LIN {X 0.050,Y -397.662,Z 1546.991,A 0.000,B 0.000,C 90.000,E1 34.358} C_DIS
LIN {X 0.138,Y -393.883,Z 1546.977,A 0.000,B 0.000,C 90.000,E1 31.878} C_DIS
LIN {X -0.084,Y -386.471,Z 1546.953,A 0.000,B 0.000,C 90.000,E1 27.641} C_DIS
LIN {X -0.108,Y -382.780,Z 1546.938,A 0.000,B 0.000,C 90.000,E1 24.771} C_DIS
LIN {X -0.152,Y -376.091,Z 1546.911,A 0.000,B 0.000,C 90.000,E1 20.066} C_DIS
LIN {X 0.190,Y -373.623,Z 1546.897,A 0.000,B 0.000,C 90.000,E1 17.457} C_DIS
LIN {X -0.137,Y -368.025,Z 1546.869,A 0.000,B 0.000,C 90.000,E1 12.355} C_DIS
LIN {X 0.096,Y -366.318,Z 1546.854,A 0.000,B 0.000,C 90.000,E1 9.726} C_DIS
LIN {X -0.025,Y -361.708,Z 1546.821,A 0.000,B 0.000,C 90.000,E1 3.784} C_DIS
LIN {X 0.055,Y -360.909,Z 1546.802,A 0.000,B 0.000,C 90.000,E1 0.401} C_DIS
LIN {X 0.137,Y -360.684,Z 1546.799,A 0.000,B 0.000,C 90.000,E1 359.771} C_DIS
LIN {X -0.053,Y -359.426,Z 1546.770,A 0.000,B 0.000,C 90.000,E1 354.546} C_DIS
LIN {X 0.070,Y -358.890,Z 1546.759,A 0.000,B 0.000,C 90.000,E1 352.648} C_DIS
LIN {X -0.020,Y -359.563,Z 1546.726,A 0.000,B 0.000,C 90.000,E1 346.645} C_DIS
LIN {X 0.001,Y -361.801,Z 1546.684,A 0.000,B 0.000,C 90.000,E1 339.135} C_DIS
LIN {X -0.154,Y -362.053,Z 1546.680,A 0.000,B 0.000,C 90.000,E1 338.411} C_DIS
LIN {X 0.189,Y -365.980,Z 1546.643,A 0.000,B 0.000,C 90.000,E1 331.641} C_DIS
LIN {X 0.029,Y -366.387,Z 1546.639,A 0.000,B 0.000,C 90.000,E1 330.923} C_DIS
LIN {X -0.031,Y -371.355,Z 1546.604,A 0.000,B 0.000,C 90.000,E1 324.642} C_DIS
LIN {X -0.043,Y -371.766,Z 1546.602,A 0.000,B 0.000,C 90.000,E1 324.276} C_DIS
LIN {X 0.013,Y -377.358,Z 1546.567,A 0.000,B 0.000,C 90.000,E1 318.038} C_DIS
LIN {X 0.012,Y -378.235,Z 1546.563,A 0.000,B 0.000,C 90.000,E1 317.310} C_DIS
LIN {X 0.002,Y -383.940,Z 1546.531,A 0.000,B 0.000,C 90.000,E1 311.515} C_DIS
LIN {X 0.088,Y -384.893,Z 1546.527,A 0.000,B 0.000,C 90.000,E1 310.782} C_DIS
LIN {X 0.262,Y -390.610,Z 1546.495,A 0.000,B 0.000,C 90.000,E1 305.025} C_DIS
LIN {X 0.106,Y -391.104,Z 1546.493,A 0.000,B 0.000,C 90.000,E1 304.692} C_DIS
LIN {X 0.022,Y -391.648,Z 1546.489,A 0.000,B 0.000,C 90.000,E1 303.992} C_DIS
LIN {X -0.080,Y -396.825,Z 1546.459,A 0.000,B 0.000,C 90.000,E1 298.693} C_DIS
LIN {X -0.210,Y -397.120,Z 1546.457,A 0.000,B 0.000,C 90.000,E1 298.359} C_DIS
LIN {X -0.055,Y -401.597,Z 1546.426,A 0.000,B 0.000,C 90.000,E1 292.717} C_DIS
LIN {X 0.222,Y -404.659,Z 1546.395,A 0.000,B 0.000,C 90.000,E1 287.094} C_DIS
LIN {X -0.079,Y -404.735,Z 1546.391,A 0.000,B 0.000,C 90.000,E1 286.441} C_DIS
LIN {X 0.214,Y -406.099,Z 1546.364,A 0.000,B 0.000,C 90.000,E1 281.535} C_DIS
LIN {X -0.176,Y -406.094,Z 1546.362,A 0.000,B 0.000,C 90.000,E1 281.243} C_DIS
LIN {X -0.097,Y -405.680,Z 1546.333,A 0.000,B 0.000,C 90.000,E1 276.024} C_DIS
LIN {X -0.165,Y -405.058,Z 1546.328,A 0.000,B 0.000,C 90.000,E1 274.992} C_DIS
LIN {X -0.060,Y -403.497,Z 1546.304,A 0.000,B 0.000,C 90.000,E1 270.802} C_DIS
LIN {X -0.092,Y -403.288,Z 1546.302,A 0.000,B 0.000,C 90.000,E1 270.458} C_DIS
LIN {X 0.091,Y -398.931,Z 1546.271,A 0.000,B 0.000,C 90.000,E1 264.837} C_DIS
LIN {X -0.040,Y -393.108,Z 1546.242,A 0.000,B 0.000,C 90.000,E1 259.567} C_DIS
LIN {X -0.079,Y -392.835,Z 1546.240,A 0.000,B 0.000,C 90.000,E1 259.218} C_DIS
LIN {X 0.034,Y -385.993,Z 1546.212,A 0.000,B 0.000,C 90.000,E1 254.212} C_DIS
LIN {X -0.026,Y -385.267,Z 1546.208,A 0.000,B 0.000,C 90.000,E1 253.504} C_DIS
LIN {X -0.004,Y -384.768,Z 1546.206,A 0.000,B 0.000,C 90.000,E1 253.142} C_DIS
LIN {X 0.221,Y -377.973,Z 1546.182,A 0.000,B 0.000,C 90.000,E1 248.773} C_DIS
LIN {X -0.044,Y -376.233,Z 1546.174,A 0.000,B 0.000,C 90.000,E1 247.358} C_DIS
LIN {X 0.057,Y -374.944,Z 1546.170,A 0.000,B 0.000,C 90.000,E1 246.613} C_DIS
LIN {X -0.208,Y -368.417,Z 1546.148,A 0.000,B 0.000,C 90.000,E1 242.615} C_DIS
LIN {X 0.097,Y -366.047,Z 1546.137,A 0.000,B 0.000,C 90.000,E1 240.717} C_DIS
LIN {X 0.004,Y -359.196,Z 1546.115,A 0.000,B 0.000,C 90.000,E1 236.628} C_DIS
LIN {X 0.021,Y -355.842,Z 1546.100,A 0.000,B 0.000,C 90.000,E1 233.989} C_DIS
LIN {X -0.173,Y -348.793,Z 1546.075,A 0.000,B 0.000,C 90.000,E1 229.461} C_DIS
LIN {X -0.097,Y -346.185,Z 1546.062,A 0.000,B 0.000,C 90.000,E1 227.148} C_DIS
LIN {X -0.088,Y -345.065,Z 1546.058,A 0.000,B 0.000,C 90.000,E1 226.377} C_DIS
LIN {X 0.094,Y -338.586,Z 1546.030,A 0.000,B 0.000,C 90.000,E1 221.310} C_DIS
LIN {X 0.094,Y -336.840,Z 1546.019,A 0.000,B 0.000,C 90.000,E1 219.358} C_DIS
LIN {X 0.014,Y -330.861,Z 1545.988,A 0.000,B 0.000,C 90.000,E1 213.865} C_DIS
LIN {X 0.149,Y -329.296,Z 1545.975,A 0.000,B 0.000,C 90.000,E1 211.465} C_DIS
LIN {X -0.154,Y -324.669,Z 1545.942,A 0.000,B 0.000,C 90.000,E1 205.540} C_DIS
LIN {X 0.174,Y -323.837,Z 1545.928,A 0.000,B 0.000,C 90.000,E1 203.078} C_DIS
LIN {X -0.017,Y -321.124,Z 1545.881,A 0.000,B 0.000,C 90.000,E1 194.662} C_DIS
LIN {X 0.138,Y -320.932,Z 1545.877,A 0.000,B 0.000,C 90.000,E1 193.828} C_DIS
LIN {X -0.076,Y -321.562,Z 1545.832,A 0.000,B 0.000,C 90.000,E1 185.796} C_DIS
LIN {X -0.143,Y -324.415,Z 1545.790,A 0.000,B 0.000,C 90.000,E1 178.165} C_DIS
LIN {X -0.141,Y -325.376,Z 1545.783,A 0.000,B 0.000,C 90.000,E1 176.963} C_DIS
LIN {X -0.100,Y -329.112,Z 1545.750,A 0.000,B 0.000,C 90.000,E1 170.971} C_DIS
LIN {X 0.061,Y -334.260,Z 1545.726,A 0.000,B 0.000,C 90.000,E1 166.589} C_DIS
LIN {X 0.067,Y -335.488,Z 1545.719,A 0.000,B 0.000,C 90.000,E1 165.408} C_DIS
LIN {X 0.143,Y -340.932,Z 1545.695,A 0.000,B 0.000,C 90.000,E1 161.094} C_DIS
LIN {X -0.172,Y -342.138,Z 1545.691,A 0.000,B 0.000,C 90.000,E1 160.369} C_DIS
LIN {X -0.058,Y -347.939,Z 1545.667,A 0.000,B 0.000,C 90.000,E1 156.102} C_DIS
LIN {X -0.081,Y -354.259,Z 1545.648,A 0.000,B 0.000,C 90.000,E1 152.666} C_DIS
LIN {X -0.222,Y -361.406,Z 1545.625,A 0.000,B 0.000,C 90.000,E1 148.535} C_DIS
LIN {X 0.065,Y -368.758,Z 1545.606,A 0.000,B 0.000,C 90.000,E1 145.135} C_DIS
LIN {X 0.065,Y -377.029,Z 1545.584,A 0.000,B 0.000,C 90.000,E1 141.090} C_DIS
LIN {X -0.061,Y -383.435,Z 1545.570,A 0.000,B 0.000,C 90.000,E1 138.566} C_DIS
LIN {X -0.015,Y -385.037,Z 1545.566,A 0.000,B 0.000,C 90.000,E1 137.838} C_DIS
LIN {X -0.004,Y -394.325,Z 1545.544,A 0.000,B 0.000,C 90.000,E1 133.905} C_DIS
LIN {X 0.107,Y -399.276,Z 1545.534,A 0.000,B 0.000,C 90.000,E1 132.123} C_DIS
LIN {X 0.210,Y -400.192,Z 1545.532,A 0.000,B 0.000,C 90.000,E1 131.757} C_DIS
LIN {X -0.113,Y -409.687,Z 1545.511,A 0.000,B 0.000,C 90.000,E1 127.971} C_DIS
LIN {X -0.007,Y -413.282,Z 1545.504,A 0.000,B 0.000,C 90.000,E1 126.710} C_DIS
LIN {X -0.059,Y -546.775,Z 1545.504,A 0.000,B 0.000,C 90.000,E1 126.710} C_DIS
LIN {X -0.108,Y -546.987,Z 1545.504,A 0.000,B 0.000,C 90.000,E1 126.710} C_DIS
LIN {X -0.068,Y -548.594,Z 1545.503,A 0.000,B 0.000,C 90.000,E1 126.583} C_DIS
LIN {X -0.261,Y -549.981,Z 1545.502,A 0.000,B 0.000,C 90.000,E1 126.377} C_DIS
LIN {X -0.211,Y -551.155,Z 1545.500,A 0.000,B 0.000,C 90.000,E1 126.091} C_DIS
LIN {X -0.155,Y -552.052,Z 1545.499,A 0.000,B 0.000,C 90.000,E1 125.804} C_DIS
LIN {X -0.032,Y -553.435,Z 1545.496,A 0.000,B 0.000,C 90.000,E1 125.231} C_DIS
LIN {X -0.218,Y -554.446,Z 1545.493,A 0.000,B 0.000,C 90.000,E1 124.692} C_DIS
LIN {X -0.079,Y -555.198,Z 1545.490,A 0.000,B 0.000,C 90.000,E1 124.119} C_DIS
LIN {X -0.175,Y -555.961,Z 1545.485,A 0.000,B 0.000,C 90.000,E1 123.293} C_DIS
LIN {X 0.204,Y -556.380,Z 1545.480,A 0.000,B 0.000,C 90.000,E1 122.418} C_DIS
LIN {X -0.259,Y -556.821,Z 1545.471,A 0.000,B 0.000,C 90.000,E1 120.797} C_DIS
LIN {X 0.241,Y -557.434,Z 1545.462,A 0.000,B 0.000,C 90.000,E1 119.077} C_DIS
LIN {X 0.151,Y -557.900,Z 1545.456,A 0.000,B 0.000,C 90.000,E1 117.975} C_DIS
LIN {X 0.151,Y -558.432,Z 1545.446,A 0.000,B 0.000,C 90.000,E1 116.309} C_DIS
LIN {X 0.068,Y -558.836,Z 1545.440,A 0.000,B 0.000,C 90.000,E1 115.207} C_DIS
LIN {X 0.044,Y -559.225,Z 1545.432,A 0.000,B 0.000,C 90.000,E1 113.823} C_DIS
LIN {X -0.195,Y -559.482,Z 1545.425,A 0.000,B 0.000,C 90.000,E1 112.461} C_DIS
LIN {X -0.227,Y -559.760,Z 1545.412,A 0.000,B 0.000,C 90.000,E1 110.248} C_DIS
LIN {X -0.124,Y -560.052,Z 1545.405,A 0.000,B 0.000,C 90.000,E1 108.852} C_DIS
LIN {X 0.115,Y -560.381,Z 1545.396,A 0.000,B 0.000,C 90.000,E1 107.166} C_DIS
LIN {X -0.048,Y -560.656,Z 1545.385,A 0.000,B 0.000,C 90.000,E1 105.245} C_DIS
LIN {X -0.114,Y -560.876,Z 1545.375,A 0.000,B 0.000,C 90.000,E1 103.592} C_DIS
LIN {X -0.143,Y -561.355,Z 1545.365,A 0.000,B 0.000,C 90.000,E1 101.658} C_DIS
LIN {X -0.107,Y -562.046,Z 1545.352,A 0.000,B 0.000,C 90.000,E1 99.443} C_DIS
LIN {X 0.025,Y -562.488,Z 1545.345,A 0.000,B 0.000,C 90.000,E1 98.049} C_DIS
LIN {X 0.233,Y -563.041,Z 1545.336,A 0.000,B 0.000,C 90.000,E1 96.372} C_DIS
LIN {X -0.179,Y -563.589,Z 1545.326,A 0.000,B 0.000,C 90.000,E1 94.759} C_DIS
LIN {X -0.070,Y -564.047,Z 1545.317,A 0.000,B 0.000,C 90.000,E1 93.094} C_DIS
LIN {X 0.021,Y -564.489,Z 1545.308,A 0.000,B 0.000,C 90.000,E1 91.432} C_DIS
LIN {X 0.115,Y -565.104,Z 1545.299,A 0.000,B 0.000,C 90.000,E1 89.771} C_DIS
LIN {X -0.214,Y -565.849,Z 1545.288,A 0.000,B 0.000,C 90.000,E1 87.879} C_DIS
LIN {X -0.078,Y -566.530,Z 1545.279,A 0.000,B 0.000,C 90.000,E1 86.216} C_DIS
LIN {X -0.274,Y -566.863,Z 1545.274,A 0.000,B 0.000,C 90.000,E1 85.412} C_DIS
LIN {X 0.230,Y -567.860,Z 1545.262,A 0.000,B 0.000,C 90.000,E1 83.166} C_DIS
LIN {X 0.175,Y -569.101,Z 1545.252,A 0.000,B 0.000,C 90.000,E1 81.254} C_DIS
LIN {X -0.037,Y -570.370,Z 1545.242,A 0.000,B 0.000,C 90.000,E1 79.634} C_DIS
LIN {X -0.213,Y -571.393,Z 1545.235,A 0.000,B 0.000,C 90.000,E1 78.285} C_DIS
LIN {X -0.172,Y -572.663,Z 1545.226,A 0.000,B 0.000,C 90.000,E1 76.645} C_DIS
LIN {X 0.190,Y -573.542,Z 1545.220,A 0.000,B 0.000,C 90.000,E1 75.519} C_DIS
LIN {X 0.207,Y -574.412,Z 1545.212,A 0.000,B 0.000,C 90.000,E1 74.157} C_DIS
LIN {X 0.038,Y -575.450,Z 1545.203,A 0.000,B 0.000,C 90.000,E1 72.543} C_DIS
LIN {X 0.052,Y -576.077,Z 1545.197,A 0.000,B 0.000,C 90.000,E1 71.456} C_DIS
LIN {X -0.080,Y -577.133,Z 1545.187,A 0.000,B 0.000,C 90.000,E1 69.571} C_DIS
LIN {X 0.014,Y -578.298,Z 1545.176,A 0.000,B 0.000,C 90.000,E1 67.667} C_DIS
LIN {X -0.179,Y -579.374,Z 1545.166,A 0.000,B 0.000,C 90.000,E1 65.793} C_DIS
LIN {X -0.109,Y -580.518,Z 1545.155,A 0.000,B 0.000,C 90.000,E1 63.896} C_DIS
LIN {X -0.273,Y -581.829,Z 1545.145,A 0.000,B 0.000,C 90.000,E1 62.025} C_DIS
LIN {X -0.131,Y -583.026,Z 1545.134,A 0.000,B 0.000,C 90.000,E1 60.127} C_DIS
LIN {X -0.169,Y -584.278,Z 1545.124,A 0.000,B 0.000,C 90.000,E1 58.250} C_DIS
LIN {X -0.228,Y -585.177,Z 1545.116,A 0.000,B 0.000,C 90.000,E1 56.914} C_DIS
LIN {X 0.181,Y -585.866,Z 1545.110,A 0.000,B 0.000,C 90.000,E1 55.801} C_DIS
LIN {X -0.215,Y -586.449,Z 1545.104,A 0.000,B 0.000,C 90.000,E1 54.769} C_DIS
LIN {X -0.073,Y -586.951,Z 1545.097,A 0.000,B 0.000,C 90.000,E1 53.417} C_DIS
LIN {X -0.120,Y -587.165,Z 1545.091,A 0.000,B 0.000,C 90.000,E1 52.351} C_DIS
LIN {X 0.001,Y -587.122,Z 1545.086,A 0.000,B 0.000,C 90.000,E1 51.537} C_DIS
LIN {X 0.123,Y -586.693,Z 1545.082,A 0.000,B 0.000,C 90.000,E1 50.723} C_DIS
LIN {X 0.053,Y -586.159,Z 1545.079,A 0.000,B 0.000,C 90.000,E1 50.194} C_DIS
LIN {X -0.019,Y -585.298,Z 1545.076,A 0.000,B 0.000,C 90.000,E1 49.666} C_DIS
LIN {X 0.166,Y -584.660,Z 1545.074,A 0.000,B 0.000,C 90.000,E1 49.380} C_DIS
LIN {X -0.096,Y -583.718,Z 1545.073,A 0.000,B 0.000,C 90.000,E1 49.138} C_DIS
LIN {X -0.198,Y -583.003,Z 1545.072,A 0.000,B 0.000,C 90.000,E1 49.013} C_DIS
LIN {X 0.083,Y -581.795,Z 1545.072,A 0.000,B 0.000,C 90.000,E1 48.852} C_DIS
LIN {X -0.287,Y -580.903,Z 1545.071,A 0.000,B 0.000,C 90.000,E1 48.852} C_DIS
LIN {X -0.235,Y -426.626,Z 1545.071,A 0.000,B 0.000,C 90.000,E1 48.852} C_DIS
LIN {X 0.007,Y -418.745,Z 1545.049,A 0.000,B 0.000,C 90.000,E1 44.879} C_DIS
LIN {X -0.027,Y -409.817,Z 1545.027,A 0.000,B 0.000,C 90.000,E1 40.782} C_DIS
LIN {X 0.010,Y -406.219,Z 1545.015,A 0.000,B 0.000,C 90.000,E1 38.705} C_DIS
LIN {X -0.163,Y -405.585,Z 1545.013,A 0.000,B 0.000,C 90.000,E1 38.382} C_DIS
LIN {X -0.100,Y -396.754,Z 1544.988,A 0.000,B 0.000,C 90.000,E1 33.833} C_DIS
LIN {X 0.209,Y -393.545,Z 1544.976,A 0.000,B 0.000,C 90.000,E1 31.671} C_DIS
LIN {X -0.039,Y -386.183,Z 1544.952,A 0.000,B 0.000,C 90.000,E1 27.436} C_DIS
LIN {X 0.108,Y -382.981,Z 1544.938,A 0.000,B 0.000,C 90.000,E1 24.899} C_DIS
LIN {X 0.089,Y -376.698,Z 1544.914,A 0.000,B 0.000,C 90.000,E1 20.556} C_DIS
LIN {X 0.071,Y -373.759,Z 1544.898,A 0.000,B 0.000,C 90.000,E1 17.638} C_DIS
LIN {X 0.019,Y -372.861,Z 1544.894,A 0.000,B 0.000,C 90.000,E1 16.913} C_DIS
LIN {X -0.079,Y -367.596,Z 1544.865,A 0.000,B 0.000,C 90.000,E1 11.771} C_DIS
LIN {X 0.006,Y -366.477,Z 1544.855,A 0.000,B 0.000,C 90.000,E1 9.905} C_DIS
LIN {X -0.057,Y -361.781,Z 1544.822,A 0.000,B 0.000,C 90.000,E1 3.955} C_DIS
LIN {X -0.172,Y -360.898,Z 1544.801,A 0.000,B 0.000,C 90.000,E1 0.229} C_DIS
LIN {X -0.053,Y -359.426,Z 1544.770,A 0.000,B 0.000,C 90.000,E1 354.546} C_DIS
LIN {X 0.070,Y -358.890,Z 1544.759,A 0.000,B 0.000,C 90.000,E1 352.648} C_DIS
LIN {X -0.020,Y -359.563,Z 1544.726,A 0.000,B 0.000,C 90.000,E1 346.645} C_DIS
LIN {X 0.001,Y -361.801,Z 1544.684,A 0.000,B 0.000,C 90.000,E1 339.135} C_DIS
LIN {X -0.154,Y -362.053,Z 1544.680,A 0.000,B 0.000,C 90.000,E1 338.411} C_DIS
LIN {X 0.189,Y -365.980,Z 1544.643,A 0.000,B 0.000,C 90.000,E1 331.641} C_DIS
LIN {X 0.029,Y -366.387,Z 1544.639,A 0.000,B 0.000,C 90.000,E1 330.923} C_DIS
LIN {X -0.031,Y -371.355,Z 1544.604,A 0.000,B 0.000,C 90.000,E1 324.642} C_DIS
LIN {X -0.043,Y -371.766,Z 1544.602,A 0.000,B 0.000,C 90.000,E1 324.276} C_DIS
LIN {X 0.013,Y -377.358,Z 1544.567,A 0.000,B 0.000,C 90.000,E1 318.038} C_DIS
LIN {X 0.012,Y -378.235,Z 1544.563,A 0.000,B 0.000,C 90.000,E1 317.310} C_DIS
LIN {X 0.002,Y -383.940,Z 1544.531,A 0.000,B 0.000,C 90.000,E1 311.515} C_DIS
LIN {X 0.088,Y -384.893,Z 1544.527,A 0.000,B 0.000,C 90.000,E1 310.782} C_DIS
LIN {X 0.262,Y -390.610,Z 1544.495,A 0.000,B 0.000,C 90.000,E1 305.025} C_DIS
LIN {X 0.106,Y -391.104,Z 1544.493,A 0.000,B 0.000,C 90.000,E1 304.692} C_DIS
LIN {X 0.022,Y -391.648,Z 1544.489,A 0.000,B 0.000,C 90.000,E1 303.992} C_DIS
LIN {X -0.080,Y -396.825,Z 1544.459,A 0.000,B 0.000,C 90.000,E1 298.693} C_DIS
LIN {X -0.210,Y -397.120,Z 1544.457,A 0.000,B 0.000,C 90.000,E1 298.359} C_DIS
LIN {X -0.055,Y -401.597,Z 1544.426,A 0.000,B 0.000,C 90.000,E1 292.717} C_DIS
LIN {X 0.222,Y -404.659,Z 1544.395,A 0.000,B 0.000,C 90.000,E1 287.094} C_DIS
LIN {X -0.079,Y -404.735,Z 1544.391,A 0.000,B 0.000,C 90.000,E1 286.441} C_DIS
LIN {X 0.214,Y -406.099,Z 1544.364,A 0.000,B 0.000,C 90.000,E1 281.535} C_DIS
LIN {X -0.176,Y -406.094,Z 1544.362,A 0.000,B 0.000,C 90.000,E1 281.243} C_DIS
LIN {X -0.097,Y -405.680,Z 1544.333,A 0.000,B 0.000,C 90.000,E1 276.024} C_DIS
LIN {X -0.165,Y -405.058,Z 1544.328,A 0.000,B 0.000,C 90.000,E1 274.992} C_DIS
LIN {X -0.060,Y -403.497,Z 1544.304,A 0.000,B 0.000,C 90.000,E1 270.802} C_DIS
LIN {X -0.092,Y -403.288,Z 1544.302,A 0.000,B 0.000,C 90.000,E1 270.458} C_DIS
LIN {X 0.091,Y -398.931,Z 1544.271,A 0.000,B 0.000,C 90.000,E1 264.837} C_DIS
LIN {X -0.040,Y -393.108,Z 1544.242,A 0.000,B 0.000,C 90.000,E1 259.567} C_DIS
LIN {X -0.079,Y -392.835,Z 1544.240,A 0.000,B 0.000,C 90.000,E1 259.218} C_DIS
LIN {X 0.034,Y -385.993,Z 1544.212,A 0.000,B 0.000,C 90.000,E1 254.212} C_DIS
LIN {X -0.026,Y -385.267,Z 1544.208,A 0.000,B 0.000,C 90.000,E1 253.504} C_DIS
LIN {X -0.004,Y -384.768,Z 1544.206,A 0.000,B 0.000,C 90.000,E1 253.142} C_DIS
LIN {X 0.221,Y -377.973,Z 1544.182,A 0.000,B 0.000,C 90.000,E1 248.773} C_DIS
LIN {X -0.044,Y -376.233,Z 1544.174,A 0.000,B 0.000,C 90.000,E1 247.358} C_DIS
LIN {X 0.057,Y -374.944,Z 1544.170,A 0.000,B 0.000,C 90.000,E1 246.613} C_DIS
LIN {X -0.208,Y -368.417,Z 1544.148,A 0.000,B 0.000,C 90.000,E1 242.615} C_DIS
LIN {X 0.097,Y -366.047,Z 1544.137,A 0.000,B 0.000,C 90.000,E1 240.717} C_DIS
LIN {X 0.004,Y -359.196,Z 1544.115,A 0.000,B 0.000,C 90.000,E1 236.628} C_DIS
LIN {X 0.021,Y -355.842,Z 1544.100,A 0.000,B 0.000,C 90.000,E1 233.989} C_DIS
LIN {X -0.173,Y -348.793,Z 1544.075,A 0.000,B 0.000,C 90.000,E1 229.461} C_DIS
LIN {X -0.097,Y -346.185,Z 1544.062,A 0.000,B 0.000,C 90.000,E1 227.148} C_DIS
LIN {X -0.088,Y -345.065,Z 1544.058,A 0.000,B 0.000,C 90.000,E1 226.377} C_DIS
LIN {X 0.094,Y -338.586,Z 1544.030,A 0.000,B 0.000,C 90.000,E1 221.310} C_DIS
LIN {X 0.094,Y -336.840,Z 1544.019,A 0.000,B 0.000,C 90.000,E1 219.358} C_DIS
LIN {X 0.014,Y -330.861,Z 1543.988,A 0.000,B 0.000,C 90.000,E1 213.865} C_DIS
LIN {X 0.149,Y -329.296,Z 1543.975,A 0.000,B 0.000,C 90.000,E1 211.465} C_DIS
LIN {X -0.154,Y -324.669,Z 1543.942,A 0.000,B 0.000,C 90.000,E1 205.540} C_DIS
LIN {X 0.174,Y -323.837,Z 1543.928,A 0.000,B 0.000,C 90.000,E1 203.078} C_DIS
LIN {X -0.017,Y -321.124,Z 1543.881,A 0.000,B 0.000,C 90.000,E1 194.662} C_DIS
LIN {X 0.138,Y -320.932,Z 1543.877,A 0.000,B 0.000,C 90.000,E1 193.828} C_DIS
LIN {X -0.076,Y -321.562,Z 1543.832,A 0.000,B 0.000,C 90.000,E1 185.796} C_DIS
LIN {X -0.143,Y -324.415,Z 1543.790,A 0.000,B 0.000,C 90.000,E1 178.165} C_DIS
LIN {X -0.141,Y -325.376,Z 1543.783,A 0.000,B 0.000,C 90.000,E1 176.963} C_DIS
LIN {X -0.100,Y -329.112,Z 1543.750,A 0.000,B 0.000,C 90.000,E1 170.971} C_DIS
LIN {X 0.061,Y -334.260,Z 1543.726,A 0.000,B 0.000,C 90.000,E1 166.589} C_DIS
LIN {X 0.067,Y -335.488,Z 1543.719,A 0.000,B 0.000,C 90.000,E1 165.408} C_DIS
LIN {X 0.143,Y -340.932,Z 1543.695,A 0.000,B 0.000,C 90.000,E1 161.094} C_DIS
LIN {X -0.172,Y -342.138,Z 1543.691,A 0.000,B 0.000,C 90.000,E1 160.369} C_DIS
LIN {X -0.058,Y -347.939,Z 1543.667,A 0.000,B 0.000,C 90.000,E1 156.102} C_DIS
LIN {X -0.081,Y -354.259,Z 1543.648,A 0.000,B 0.000,C 90.000,E1 152.666} C_DIS
LIN {X -0.222,Y -361.406,Z 1543.625,A 0.000,B 0.000,C 90.000,E1 148.535} C_DIS
LIN {X 0.065,Y -368.758,Z 1543.606,A 0.000,B 0.000,C 90.000,E1 145.135} C_DIS
LIN {X 0.065,Y -377.029,Z 1543.584,A 0.000,B 0.000,C 90.000,E1 141.090} C_DIS
LIN {X -0.061,Y -383.435,Z 1543.570,A 0.000,B 0.000,C 90.000,E1 138.566} C_DIS
LIN {X -0.015,Y -385.037,Z 1543.566,A 0.000,B 0.000,C 90.000,E1 137.838} C_DIS
LIN {X -0.004,Y -394.325,Z 1543.544,A 0.000,B 0.000,C 90.000,E1 133.905} C_DIS
LIN {X 0.107,Y -399.276,Z 1543.534,A 0.000,B 0.000,C 90.000,E1 132.123} C_DIS
LIN {X 0.210,Y -400.192,Z 1543.532,A 0.000,B 0.000,C 90.000,E1 131.757} C_DIS
LIN {X 0.128,Y -410.042,Z 1543.510,A 0.000,B 0.000,C 90.000,E1 127.810} C_DIS
LIN {X 0.030,Y -410.207,Z 1543.510,A 0.000,B 0.000,C 90.000,E1 127.764} C_DIS
LIN {X 0.346,Y -546.218,Z 1543.510,A 0.000,B 0.000,C 90.000,E1 127.729} C_DIS
LIN {X 0.260,Y -546.637,Z 1543.510,A 0.000,B 0.000,C 90.000,E1 127.729} C_DIS
LIN {X 0.055,Y -548.450,Z 1543.509,A 0.000,B 0.000,C 90.000,E1 127.604} C_DIS
LIN {X 0.098,Y -549.852,Z 1543.508,A 0.000,B 0.000,C 90.000,E1 127.363} C_DIS
LIN {X 0.148,Y -551.009,Z 1543.506,A 0.000,B 0.000,C 90.000,E1 127.076} C_DIS
LIN {X 0.203,Y -551.924,Z 1543.505,A 0.000,B 0.000,C 90.000,E1 126.790} C_DIS
LIN {X 0.263,Y -552.678,Z 1543.503,A 0.000,B 0.000,C 90.000,E1 126.503} C_DIS
LIN {X 0.066,Y -553.840,Z 1543.500,A 0.000,B 0.000,C 90.000,E1 125.964} C_DIS
LIN {X 0.278,Y -555.128,Z 1543.495,A 0.000,B 0.000,C 90.000,E1 125.105} C_DIS
LIN {X 0.183,Y -555.983,Z 1543.491,A 0.000,B 0.000,C 90.000,E1 124.278} C_DIS
LIN {X 0.100,Y -556.458,Z 1543.486,A 0.000,B 0.000,C 90.000,E1 123.452} C_DIS
LIN {X -0.132,Y -556.796,Z 1543.478,A 0.000,B 0.000,C 90.000,E1 122.084} C_DIS
LIN {X 0.287,Y -557.534,Z 1543.464,A 0.000,B 0.000,C 90.000,E1 119.539} C_DIS
LIN {X -0.012,Y -558.101,Z 1543.457,A 0.000,B 0.000,C 90.000,E1 118.180} C_DIS
LIN {X 0.247,Y -558.604,Z 1543.447,A 0.000,B 0.000,C 90.000,E1 116.488} C_DIS
LIN {X -0.077,Y -558.995,Z 1543.441,A 0.000,B 0.000,C 90.000,E1 115.412} C_DIS
LIN {X -0.091,Y -559.388,Z 1543.433,A 0.000,B 0.000,C 90.000,E1 114.027} C_DIS
LIN {X 0.203,Y -559.665,Z 1543.424,A 0.000,B 0.000,C 90.000,E1 112.333} C_DIS
LIN {X -0.134,Y -559.924,Z 1543.413,A 0.000,B 0.000,C 90.000,E1 110.429} C_DIS
LIN {X 0.276,Y -560.259,Z 1543.404,A 0.000,B 0.000,C 90.000,E1 108.725} C_DIS
LIN {X 0.115,Y -560.593,Z 1543.393,A 0.000,B 0.000,C 90.000,E1 106.804} C_DIS
LIN {X -0.195,Y -560.887,Z 1543.383,A 0.000,B 0.000,C 90.000,E1 104.898} C_DIS
LIN {X 0.183,Y -561.272,Z 1543.370,A 0.000,B 0.000,C 90.000,E1 102.647} C_DIS
LIN {X 0.244,Y -561.570,Z 1543.364,A 0.000,B 0.000,C 90.000,E1 101.535} C_DIS
LIN {X 0.275,Y -562.282,Z 1543.352,A 0.000,B 0.000,C 90.000,E1 99.321} C_DIS
LIN {X -0.233,Y -562.728,Z 1543.344,A 0.000,B 0.000,C 90.000,E1 97.992} C_DIS
LIN {X -0.018,Y -563.313,Z 1543.335,A 0.000,B 0.000,C 90.000,E1 96.315} C_DIS
LIN {X 0.139,Y -563.875,Z 1543.326,A 0.000,B 0.000,C 90.000,E1 94.645} C_DIS
LIN {X 0.256,Y -564.302,Z 1543.317,A 0.000,B 0.000,C 90.000,E1 92.980} C_DIS
LIN {X 0.247,Y -564.742,Z 1543.309,A 0.000,B 0.000,C 90.000,E1 91.604} C_DIS
LIN {X -0.108,Y -565.453,Z 1543.298,A 0.000,B 0.000,C 90.000,E1 89.714} C_DIS
LIN {X 0.250,Y -566.354,Z 1543.286,A 0.000,B 0.000,C 90.000,E1 87.478} C_DIS
LIN {X -0.024,Y -567.174,Z 1543.276,A 0.000,B 0.000,C 90.000,E1 85.584} C_DIS
LIN {X -0.070,Y -568.112,Z 1543.263,A 0.000,B 0.000,C 90.000,E1 83.394} C_DIS
LIN {X 0.093,Y -568.943,Z 1543.256,A 0.000,B 0.000,C 90.000,E1 82.008} C_DIS
LIN {X 0.068,Y -570.373,Z 1543.245,A 0.000,B 0.000,C 90.000,E1 80.095} C_DIS
LIN {X -0.024,Y -571.674,Z 1543.236,A 0.000,B 0.000,C 90.000,E1 78.465} C_DIS
LIN {X 0.211,Y -573.108,Z 1543.225,A 0.000,B 0.000,C 90.000,E1 76.533} C_DIS
LIN {X 0.215,Y -574.170,Z 1543.218,A 0.000,B 0.000,C 90.000,E1 75.172} C_DIS
LIN {X 0.038,Y -575.235,Z 1543.209,A 0.000,B 0.000,C 90.000,E1 73.559} C_DIS
LIN {X -0.118,Y -576.245,Z 1543.200,A 0.000,B 0.000,C 90.000,E1 71.945} C_DIS
LIN {X 0.129,Y -577.486,Z 1543.188,A 0.000,B 0.000,C 90.000,E1 69.752} C_DIS
LIN {X 0.235,Y -578.602,Z 1543.177,A 0.000,B 0.000,C 90.000,E1 67.847} C_DIS
LIN {X 0.054,Y -579.641,Z 1543.167,A 0.000,B 0.000,C 90.000,E1 65.973} C_DIS
LIN {X 0.003,Y -580.950,Z 1543.155,A 0.000,B 0.000,C 90.000,E1 63.819} C_DIS
LIN {X -0.143,Y -582.247,Z 1543.144,A 0.000,B 0.000,C 90.000,E1 61.948} C_DIS
LIN {X 0.018,Y -583.455,Z 1543.134,A 0.000,B 0.000,C 90.000,E1 60.049} C_DIS
LIN {X -0.311,Y -584.716,Z 1543.123,A 0.000,B 0.000,C 90.000,E1 58.201} C_DIS
LIN {X -0.049,Y -585.617,Z 1543.116,A 0.000,B 0.000,C 90.000,E1 56.834} C_DIS
LIN {X 0.041,Y -586.323,Z 1543.110,A 0.000,B 0.000,C 90.000,E1 55.754} C_DIS
LIN {X -0.017,Y -586.937,Z 1543.104,A 0.000,B 0.000,C 90.000,E1 54.689} C_DIS
LIN {X 0.333,Y -587.532,Z 1543.095,A 0.000,B 0.000,C 90.000,E1 53.050} C_DIS
LIN {X 0.227,Y -587.973,Z 1543.086,A 0.000,B 0.000,C 90.000,E1 51.457} C_DIS
LIN {X -0.013,Y -587.960,Z 1543.082,A 0.000,B 0.000,C 90.000,E1 50.678} C_DIS
LIN {X -0.336,Y -587.650,Z 1543.077,A 0.000,B 0.000,C 90.000,E1 49.908} C_DIS
LIN {X 0.046,Y -587.236,Z 1543.074,A 0.000,B 0.000,C 90.000,E1 49.337} C_DIS
LIN {X 0.363,Y -586.461,Z 1543.071,A 0.000,B 0.000,C 90.000,E1 48.771} C_DIS
LIN {X 0.108,Y -585.925,Z 1543.070,A 0.000,B 0.000,C 90.000,E1 48.528} C_DIS
LIN {X 0.290,Y -585.195,Z 1543.068,A 0.000,B 0.000,C 90.000,E1 48.243} C_DIS
LIN {X -0.251,Y -584.651,Z 1543.068,A 0.000,B 0.000,C 90.000,E1 48.162} C_DIS
LIN {X 0.258,Y -583.566,Z 1543.066,A 0.000,B 0.000,C 90.000,E1 47.919} C_DIS
LIN {X 0.068,Y -582.636,Z 1543.066,A 0.000,B 0.000,C 90.000,E1 47.838} C_DIS
LIN {X 0.038,Y -581.751,Z 1543.066,A 0.000,B 0.000,C 90.000,E1 47.796} C_DIS
LIN {X 0.005,Y -581.607,Z 1543.066,A 0.000,B 0.000,C 90.000,E1 47.796} C_DIS
LIN {X -0.020,Y -424.345,Z 1543.066,A 0.000,B 0.000,C 90.000,E1 47.796} C_DIS
LIN {X -0.061,Y -419.007,Z 1543.050,A 0.000,B 0.000,C 90.000,E1 45.040} C_DIS
LIN {X 0.124,Y -418.337,Z 1543.048,A 0.000,B 0.000,C 90.000,E1 44.676} C_DIS
LIN {X -0.067,Y -408.831,Z 1543.024,A 0.000,B 0.000,C 90.000,E1 40.253} C_DIS
LIN {X -0.199,Y -405.916,Z 1543.014,A 0.000,B 0.000,C 90.000,E1 38.543} C_DIS
LIN {X 0.019,Y -397.600,Z 1542.991,A 0.000,B 0.000,C 90.000,E1 34.326} C_DIS
LIN {X -0.115,Y -393.833,Z 1542.977,A 0.000,B 0.000,C 90.000,E1 31.878} C_DIS
LIN {X 0.006,Y -386.417,Z 1542.953,A 0.000,B 0.000,C 90.000,E1 27.590} C_DIS
LIN {X -0.011,Y -382.716,Z 1542.937,A 0.000,B 0.000,C 90.000,E1 24.719} C_DIS
LIN {X 0.080,Y -376.048,Z 1542.911,A 0.000,B 0.000,C 90.000,E1 19.993} C_DIS
LIN {X -0.060,Y -373.582,Z 1542.897,A 0.000,B 0.000,C 90.000,E1 17.457} C_DIS
LIN {X -0.026,Y -367.994,Z 1542.868,A 0.000,B 0.000,C 90.000,E1 12.299} C_DIS
LIN {X -0.008,Y -366.562,Z 1542.856,A 0.000,B 0.000,C 90.000,E1 10.074} C_DIS
LIN {X 0.065,Y -365.867,Z 1542.852,A 0.000,B 0.000,C 90.000,E1 9.321} C_DIS
LIN {X 0.079,Y -361.406,Z 1542.817,A 0.000,B 0.000,C 90.000,E1 2.980} C_DIS
LIN {X 0.169,Y -360.908,Z 1542.802,A 0.000,B 0.000,C 90.000,E1 0.344} C_DIS
LIN {X -0.058,Y -360.492,Z 1542.797,A 0.000,B 0.000,C 90.000,E1 359.427} C_DIS
LIN {X -0.053,Y -359.426,Z 1542.770,A 0.000,B 0.000,C 90.000,E1 354.546} C_DIS
LIN {X 0.070,Y -358.890,Z 1542.759,A 0.000,B 0.000,C 90.000,E1 352.648} C_DIS
LIN {X -0.020,Y -359.563,Z 1542.726,A 0.000,B 0.000,C 90.000,E1 346.645} C_DIS
LIN {X 0.001,Y -361.801,Z 1542.684,A 0.000,B 0.000,C 90.000,E1 339.135} C_DIS
LIN {X -0.154,Y -362.053,Z 1542.680,A 0.000,B 0.000,C 90.000,E1 338.411} C_DIS
LIN {X 0.189,Y -365.980,Z 1542.643,A 0.000,B 0.000,C 90.000,E1 331.641} C_DIS
LIN {X 0.029,Y -366.387,Z 1542.639,A 0.000,B 0.000,C 90.000,E1 330.923} C_DIS
LIN {X -0.031,Y -371.355,Z 1542.604,A 0.000,B 0.000,C 90.000,E1 324.642} C_DIS
LIN {X -0.043,Y -371.766,Z 1542.602,A 0.000,B 0.000,C 90.000,E1 324.276} C_DIS
LIN {X 0.013,Y -377.358,Z 1542.567,A 0.000,B 0.000,C 90.000,E1 318.038} C_DIS
LIN {X 0.012,Y -378.235,Z 1542.563,A 0.000,B 0.000,C 90.000,E1 317.310} C_DIS
LIN {X 0.002,Y -383.940,Z 1542.531,A 0.000,B 0.000,C 90.000,E1 311.515} C_DIS
LIN {X 0.088,Y -384.893,Z 1542.527,A 0.000,B 0.000,C 90.000,E1 310.782} C_DIS
LIN {X 0.262,Y -390.610,Z 1542.495,A 0.000,B 0.000,C 90.000,E1 305.025} C_DIS
LIN {X 0.106,Y -391.104,Z 1542.493,A 0.000,B 0.000,C 90.000,E1 304.692} C_DIS
LIN {X 0.022,Y -391.648,Z 1542.489,A 0.000,B 0.000,C 90.000,E1 303.992} C_DIS
LIN {X -0.080,Y -396.825,Z 1542.459,A 0.000,B 0.000,C 90.000,E1 298.693} C_DIS
LIN {X -0.210,Y -397.120,Z 1542.457,A 0.000,B 0.000,C 90.000,E1 298.359} C_DIS
LIN {X -0.055,Y -401.597,Z 1542.426,A 0.000,B 0.000,C 90.000,E1 292.717} C_DIS
LIN {X 0.222,Y -404.659,Z 1542.395,A 0.000,B 0.000,C 90.000,E1 287.094} C_DIS
LIN {X -0.079,Y -404.735,Z 1542.391,A 0.000,B 0.000,C 90.000,E1 286.441} C_DIS
LIN {X 0.214,Y -406.099,Z 1542.364,A 0.000,B 0.000,C 90.000,E1 281.535} C_DIS
LIN {X -0.176,Y -406.094,Z 1542.362,A 0.000,B 0.000,C 90.000,E1 281.243} C_DIS
LIN {X -0.097,Y -405.680,Z 1542.333,A 0.000,B 0.000,C 90.000,E1 276.024} C_DIS
LIN {X -0.165,Y -405.058,Z 1542.328,A 0.000,B 0.000,C 90.000,E1 274.992} C_DIS
LIN {X -0.060,Y -403.497,Z 1542.304,A 0.000,B 0.000,C 90.000,E1 270.802} C_DIS
LIN {X -0.092,Y -403.288,Z 1542.302,A 0.000,B 0.000,C 90.000,E1 270.458} C_DIS
LIN {X 0.091,Y -398.931,Z 1542.271,A 0.000,B 0.000,C 90.000,E1 264.837} C_DIS
LIN {X -0.040,Y -393.108,Z 1542.242,A 0.000,B 0.000,C 90.000,E1 259.567} C_DIS
LIN {X -0.079,Y -392.835,Z 1542.240,A 0.000,B 0.000,C 90.000,E1 259.218} C_DIS
LIN {X 0.034,Y -385.993,Z 1542.212,A 0.000,B 0.000,C 90.000,E1 254.212} C_DIS
LIN {X -0.026,Y -385.267,Z 1542.208,A 0.000,B 0.000,C 90.000,E1 253.504} C_DIS
LIN {X -0.004,Y -384.768,Z 1542.206,A 0.000,B 0.000,C 90.000,E1 253.142} C_DIS
LIN {X 0.221,Y -377.973,Z 1542.182,A 0.000,B 0.000,C 90.000,E1 248.773} C_DIS
LIN {X -0.044,Y -376.233,Z 1542.174,A 0.000,B 0.000,C 90.000,E1 247.358} C_DIS
LIN {X 0.057,Y -374.944,Z 1542.170,A 0.000,B 0.000,C 90.000,E1 246.613} C_DIS
LIN {X -0.208,Y -368.417,Z 1542.148,A 0.000,B 0.000,C 90.000,E1 242.615} C_DIS
LIN {X 0.097,Y -366.047,Z 1542.137,A 0.000,B 0.000,C 90.000,E1 240.717} C_DIS
LIN {X 0.004,Y -359.196,Z 1542.115,A 0.000,B 0.000,C 90.000,E1 236.628} C_DIS
LIN {X 0.021,Y -355.842,Z 1542.100,A 0.000,B 0.000,C 90.000,E1 233.989} C_DIS
LIN {X -0.173,Y -348.793,Z 1542.075,A 0.000,B 0.000,C 90.000,E1 229.461} C_DIS
LIN {X -0.097,Y -346.185,Z 1542.062,A 0.000,B 0.000,C 90.000,E1 227.148} C_DIS
LIN {X -0.088,Y -345.065,Z 1542.058,A 0.000,B 0.000,C 90.000,E1 226.377} C_DIS
LIN {X 0.094,Y -338.586,Z 1542.030,A 0.000,B 0.000,C 90.000,E1 221.310} C_DIS
LIN {X 0.094,Y -336.840,Z 1542.019,A 0.000,B 0.000,C 90.000,E1 219.358} C_DIS
LIN {X 0.014,Y -330.861,Z 1541.988,A 0.000,B 0.000,C 90.000,E1 213.865} C_DIS
LIN {X 0.149,Y -329.296,Z 1541.975,A 0.000,B 0.000,C 90.000,E1 211.465} C_DIS
LIN {X -0.154,Y -324.669,Z 1541.942,A 0.000,B 0.000,C 90.000,E1 205.540} C_DIS
LIN {X 0.174,Y -323.837,Z 1541.928,A 0.000,B 0.000,C 90.000,E1 203.078} C_DIS
LIN {X -0.017,Y -321.124,Z 1541.881,A 0.000,B 0.000,C 90.000,E1 194.662} C_DIS
LIN {X 0.138,Y -320.932,Z 1541.877,A 0.000,B 0.000,C 90.000,E1 193.828} C_DIS
LIN {X -0.076,Y -321.562,Z 1541.832,A 0.000,B 0.000,C 90.000,E1 185.796} C_DIS
LIN {X -0.143,Y -324.415,Z 1541.790,A 0.000,B 0.000,C 90.000,E1 178.165} C_DIS
LIN {X -0.141,Y -325.376,Z 1541.783,A 0.000,B 0.000,C 90.000,E1 176.963} C_DIS
LIN {X -0.100,Y -329.112,Z 1541.750,A 0.000,B 0.000,C 90.000,E1 170.971} C_DIS
LIN {X 0.061,Y -334.260,Z 1541.726,A 0.000,B 0.000,C 90.000,E1 166.589} C_DIS
LIN {X 0.067,Y -335.488,Z 1541.719,A 0.000,B 0.000,C 90.000,E1 165.408} C_DIS
LIN {X 0.143,Y -340.932,Z 1541.695,A 0.000,B 0.000,C 90.000,E1 161.094} C_DIS
LIN {X -0.172,Y -342.138,Z 1541.691,A 0.000,B 0.000,C 90.000,E1 160.369} C_DIS
LIN {X -0.058,Y -347.939,Z 1541.667,A 0.000,B 0.000,C 90.000,E1 156.102} C_DIS
LIN {X -0.081,Y -354.259,Z 1541.648,A 0.000,B 0.000,C 90.000,E1 152.666} C_DIS
LIN {X -0.222,Y -361.406,Z 1541.625,A 0.000,B 0.000,C 90.000,E1 148.535} C_DIS
LIN {X 0.065,Y -368.758,Z 1541.606,A 0.000,B 0.000,C 90.000,E1 145.135} C_DIS
LIN {X 0.065,Y -377.029,Z 1541.584,A 0.000,B 0.000,C 90.000,E1 141.090} C_DIS
LIN {X -0.061,Y -383.435,Z 1541.570,A 0.000,B 0.000,C 90.000,E1 138.566} C_DIS
LIN {X -0.015,Y -385.037,Z 1541.566,A 0.000,B 0.000,C 90.000,E1 137.838} C_DIS
LIN {X -0.004,Y -394.325,Z 1541.544,A 0.000,B 0.000,C 90.000,E1 133.905} C_DIS
LIN {X 0.107,Y -399.276,Z 1541.534,A 0.000,B 0.000,C 90.000,E1 132.123} C_DIS
LIN {X 0.210,Y -400.192,Z 1541.532,A 0.000,B 0.000,C 90.000,E1 131.757} C_DIS
LIN {X -0.164,Y -407.376,Z 1541.516,A 0.000,B 0.000,C 90.000,E1 128.830} C_DIS
LIN {X -0.248,Y -545.932,Z 1541.516,A 0.000,B 0.000,C 90.000,E1 128.830} C_DIS
LIN {X -0.306,Y -546.198,Z 1541.516,A 0.000,B 0.000,C 90.000,E1 128.830} C_DIS
LIN {X -0.207,Y -548.091,Z 1541.515,A 0.000,B 0.000,C 90.000,E1 128.669} C_DIS
LIN {X 0.298,Y -549.505,Z 1541.513,A 0.000,B 0.000,C 90.000,E1 128.382} C_DIS
LIN {X 0.346,Y -550.665,Z 1541.512,A 0.000,B 0.000,C 90.000,E1 128.096} C_DIS
LIN {X -0.034,Y -551.573,Z 1541.510,A 0.000,B 0.000,C 90.000,E1 127.855} C_DIS
LIN {X 0.084,Y -552.995,Z 1541.507,A 0.000,B 0.000,C 90.000,E1 127.282} C_DIS
LIN {X -0.118,Y -554.085,Z 1541.504,A 0.000,B 0.000,C 90.000,E1 126.744} C_DIS
LIN {X 0.098,Y -555.233,Z 1541.500,A 0.000,B 0.000,C 90.000,E1 125.884} C_DIS
LIN {X 0.323,Y -556.034,Z 1541.495,A 0.000,B 0.000,C 90.000,E1 125.025} C_DIS
